KUKA KRL program: EPS_2_25748_MH04A_A_20260121065900.src

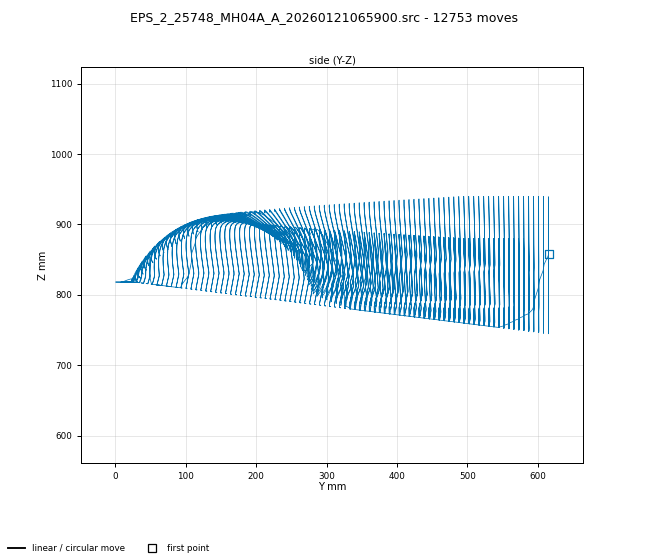
[picture p0: tool path of EPS_2_25748_MH04A_A_20260121065900.src, 12753 of 12755 moves have a stored position in this frame; points joined in program order, loops and branches not executed]
&ACCESS RVP
&REL 4
&COMMENT QRS 19112012
&PARAM EDITMASK = *
DEF PART()
EXT BAS (BAS_COMMAND :IN,REAL :IN )
INT I
BAS (#INITMOV,0 )

;KUKA QRS Post kuka4.cps  Date:22-06-2017 !

File_ID=3002

QRS_PRE_INIT()

;Init var - Until changes are made in qrs_pre_init
Outlet_Square_prg=0
Inlet_1_Square_prg=0
Inlet_2_Square_prg=0
Inlet_3_Square_prg=0
Inlet_4_Square_prg=0
Inlet_5_Square_prg=0

Outlet_1={X 0.000, Y 493.160, Z 839.500, B 0.000, E1 0.000 }
Inlet_1={X 0.000, Y 497.530, Z 779.500, B 0.000, E1 90.000 }
Inlet_2={X 0.000, Y 497.530, Z 779.500, B 0.000, E1 270.000 }
Outlet_1_type=201
Inlet_1_type=201
Inlet_2_type=201
;QRS#1=Sidecore dimensions
;QRS#2=200-8" PVC SDR 35
;QRS#3=200-8" PVC SDR 35
;QRS#4=200-8" PVC SDR 35
;QRS#5=
;QRS#6=
;QRS#7=
;QRS#8=
;QRS#9=12-08 PSX
;QRS#10=12-08 PSX
;QRS#11=12-08 PSX
;QRS#12=
;QRS#13=
;QRS#14=
;QRS#15=
;QRS#16=1220x127x1219 4'
;QRS#17=EPS Height
;QRS#18=940
;QRS#19=*
;QRS#20= UPDATED VERSION 22-06-2017
;QRS#21=*
Outlet_Square=0100
Inlet_1_Square=0100
Inlet_2_Square=0100
Inlet_3_Square=0
Inlet_4_Square=0
Inlet_5_Square=0
Mill_Square=1
Outlet_Square_Prg=204
Inlet_1_Square_prg=204
Inlet_2_Square_prg=204

QRS_INIT()

$ADVANCE=5

; T1
PTP {E1 173.418,E2 173.418}
PTP {X 0,Y 615.496,A -85,B 0,C 180,E1 173.418,E2 173.418,E3 0,E4 0,E5 0,E6 0}
QRS_SPEED_INIT()
LIN {X 0,Y 615.496,Z 858.208,A -85,B 0,C 180,E1 173.418,E2 173.418,E3 0,E4 0,E5 0,E6 0} C_VEL
LIN {X 0,Y 615.497,Z 850.543,A -85,B 0,C 180,E1 172.455,E2 172.455} C_VEL
LIN {X 0,Y 615.498,Z 840.767,A -85,B 0,C 180,E1 171.464,E2 171.464} C_VEL
LIN {X 0,Y 615.498,Z 830.503,A -85,B 0,C 180,E1 170.636,E2 170.636} C_VEL
LIN {X 0,Y 615.496,Z 818.942,A -85,B 0,C 180,E1 169.89,E2 169.89} C_VEL
LIN {X 0,Y 615.451,Z 807.364,A -85,B 0,C 180,E1 169.304,E2 169.304} C_VEL
LIN {X 0,Y 615.447,Z 795.462,A -85,B 0,C 180,E1 168.848,E2 168.848} C_VEL
LIN {X 0,Y 615.479,Z 783.419,A -85,B 0,C 180,E1 168.516,E2 168.516} C_VEL
LIN {X 0,Y 615.492,Z 776.192,A -85,B 0,C 180,E1 168.37,E2 168.37} C_VEL
LIN {X 0,Y 615.47,Z 772.045,A -85,B 0,C 180,E1 165.451,E2 165.451} C_VEL
LIN {X 0,Y 615.475,Z 768.231,A -85,B 0,C 180,E1 162.73,E2 162.73} C_VEL
LIN {X 0,Y 615.494,Z 764.414,A -85,B 0,C 180,E1 159.968,E2 159.968} C_VEL
LIN {X 0,Y 615.496,Z 761.258,A -85,B 0,C 180,E1 157.653,E2 157.653} C_VEL
LIN {X 0,Y 615.471,Z 757.73,A -85,B 0,C 180,E1 155.008,E2 155.008} C_VEL
LIN {X 0,Y 615.479,Z 754.866,A -85,B 0,C 180,E1 152.823,E2 152.823} C_VEL
LIN {X 0,Y 615.474,Z 751.515,A -85,B 0,C 180,E1 150.208,E2 150.208} C_VEL
LIN {X 0,Y 615.499,Z 748.171,A -85,B 0,C 180,E1 147.544,E2 147.544} C_VEL
LIN {X 0,Y 615.496,Z 745.306,A -85,B 0,C 180,E1 145.187,E2 145.187} C_VEL
LIN {X 0,Y 615.457,Z 744.691,A -85,B 0,C 180,E1 144.171,E2 144.171} C_VEL
LIN {X 0,Y 615.461,Z 744.688,A -85,B 0,C 180,E1 141.931,E2 141.931} C_VEL
LIN {X 0,Y 615.487,Z 744.683,A -85,B 0,C 180,E1 139.395,E2 139.395} C_VEL
LIN {X 0,Y 615.495,Z 744.698,A -85,B 0,C 180,E1 136.757,E2 136.757} C_VEL
LIN {X 0,Y 615.452,Z 744.692,A -85,B 0,C 180,E1 133.995,E2 133.995} C_VEL
LIN {X 0,Y 615.465,Z 744.686,A -85,B 0,C 180,E1 131.476,E2 131.476} C_VEL
LIN {X 0,Y 615.498,Z 744.688,A -85,B 0,C 180,E1 128.904,E2 128.904} C_VEL
LIN {X 0,Y 615.478,Z 744.701,A -85,B 0,C 180,E1 126.426,E2 126.426} C_VEL
LIN {X 0,Y 615.453,Z 744.696,A -85,B 0,C 180,E1 124.024,E2 124.024} C_VEL
LIN {X 0,Y 615.441,Z 744.693,A -85,B 0,C 180,E1 121.688,E2 121.688} C_VEL
LIN {X 0,Y 615.44,Z 744.692,A -85,B 0,C 180,E1 119.409,E2 119.409} C_VEL
LIN {X 0,Y 615.46,Z 744.69,A -85,B 0,C 180,E1 117.042,E2 117.042} C_VEL
LIN {X 0,Y 615.458,Z 744.698,A -85,B 0,C 180,E1 114.005,E2 114.005} C_VEL
LIN {X 0,Y 615.431,Z 744.694,A -85,B 0,C 180,E1 111.434,E2 111.434} C_VEL
LIN {X 0,Y 615.429,Z 744.695,A -85,B 0,C 180,E1 109.34,E2 109.34} C_VEL
LIN {X 0,Y 615.475,Z 744.692,A -85,B 0,C 180,E1 106.587,E2 106.587} C_VEL
LIN {X 0,Y 615.458,Z 744.699,A -85,B 0,C 180,E1 103.875,E2 103.875} C_VEL
LIN {X 0,Y 615.42,Z 744.697,A -85,B 0,C 180,E1 101.194,E2 101.194} C_VEL
LIN {X 0,Y 615.455,Z 744.695,A -85,B 0,C 180,E1 98.537,E2 98.537} C_VEL
LIN {X 0,Y 615.475,Z 744.7,A -85,B 0,C 180,E1 95.899,E2 95.899} C_VEL
LIN {X 0,Y 615.416,Z 744.699,A -85,B 0,C 180,E1 93.273,E2 93.273} C_VEL
LIN {X 0,Y 615.418,Z 744.699,A -85,B 0,C 180,E1 91.309,E2 91.309} C_VEL
LIN {X 0,Y 615.421,Z 744.7,A -85,B 0,C 180,E1 89.346,E2 89.346} C_VEL
LIN {X 0,Y 615.426,Z 744.7,A -85,B 0,C 180,E1 87.382,E2 87.382} C_VEL
LIN {X 0,Y 615.432,Z 744.7,A -85,B 0,C 180,E1 85.415,E2 85.415} C_VEL
LIN {X 0,Y 615.442,Z 744.699,A -85,B 0,C 180,E1 83.443,E2 83.443} C_VEL
LIN {X 0,Y 615.41,Z 744.699,A -85,B 0,C 180,E1 80.8,E2 80.8} C_VEL
LIN {X 0,Y 615.412,Z 744.698,A -85,B 0,C 180,E1 78.805,E2 78.805} C_VEL
LIN {X 0,Y 615.415,Z 744.698,A -85,B 0,C 180,E1 76.797,E2 76.797} C_VEL
LIN {X 0,Y 615.418,Z 744.697,A -85,B 0,C 180,E1 74.772,E2 74.772} C_VEL
LIN {X 0,Y 615.42,Z 744.696,A -85,B 0,C 180,E1 72.727,E2 72.727} C_VEL
LIN {X 0,Y 615.422,Z 744.696,A -85,B 0,C 180,E1 70.66,E2 70.66} C_VEL
LIN {X 0,Y 615.422,Z 744.696,A -85,B 0,C 180,E1 68.566,E2 68.566} C_VEL
LIN {X 0,Y 615.446,Z 744.698,A -85,B 0,C 180,E1 65.998,E2 65.998} C_VEL
LIN {X 0,Y 615.458,Z 744.692,A -85,B 0,C 180,E1 62.958,E2 62.958} C_VEL
LIN {X 0,Y 615.438,Z 744.693,A -85,B 0,C 180,E1 60.591,E2 60.591} C_VEL
LIN {X 0,Y 615.434,Z 744.694,A -85,B 0,C 180,E1 58.311,E2 58.311} C_VEL
LIN {X 0,Y 615.441,Z 744.696,A -85,B 0,C 180,E1 55.975,E2 55.975} C_VEL
LIN {X 0,Y 615.497,Z 744.689,A -85,B 0,C 180,E1 53.061,E2 53.061} C_VEL
LIN {X 0,Y 615.443,Z 744.691,A -85,B 0,C 180,E1 50.246,E2 50.246} C_VEL
LIN {X 0,Y 615.461,Z 744.697,A -85,B 0,C 180,E1 47.645,E2 47.645} C_VEL
LIN {X 0,Y 615.497,Z 744.689,A -85,B 0,C 180,E1 44.932,E2 44.932} C_VEL
LIN {X 0,Y 615.465,Z 744.687,A -85,B 0,C 180,E1 42.354,E2 42.354} C_VEL
LIN {X 0,Y 615.453,Z 744.693,A -85,B 0,C 180,E1 39.752,E2 39.752} C_VEL
LIN {X 0,Y 615.492,Z 744.694,A -85,B 0,C 180,E1 36.937,E2 36.937} C_VEL
LIN {X 0,Y 615.458,Z 744.693,A -85,B 0,C 180,E1 35.617,E2 35.617} C_VEL
LIN {X 0,Y 615.494,Z 745.333,A -85,B 0,C 180,E1 34.701,E2 34.701} C_VEL
LIN {X 0,Y 615.492,Z 748.215,A -85,B 0,C 180,E1 32.331,E2 32.331} C_VEL
LIN {X 0,Y 615.47,Z 751.401,A -85,B 0,C 180,E1 29.791,E2 29.791} C_VEL
LIN {X 0,Y 615.486,Z 754.919,A -85,B 0,C 180,E1 27.044,E2 27.044} C_VEL
LIN {X 0,Y 615.495,Z 758.56,A -85,B 0,C 180,E1 24.271,E2 24.271} C_VEL
LIN {X 0,Y 615.492,Z 762.386,A -85,B 0,C 180,E1 21.431,E2 21.431} C_VEL
LIN {X 0,Y 615.476,Z 766.256,A -85,B 0,C 180,E1 18.601,E2 18.601} C_VEL
LIN {X 0,Y 615.492,Z 770.016,A -85,B 0,C 180,E1 15.904,E2 15.904} C_VEL
LIN {X 0,Y 615.469,Z 773.827,A -85,B 0,C 180,E1 13.201,E2 13.201} C_VEL
LIN {X 0,Y 615.49,Z 776.183,A -85,B 0,C 180,E1 11.547,E2 11.547} C_VEL
LIN {X 0,Y 615.462,Z 791.288,A -85,B 0,C 180,E1 11.193,E2 11.193} C_VEL
LIN {X 0,Y 615.447,Z 803.206,A -85,B 0,C 180,E1 10.782,E2 10.782} C_VEL
LIN {X 0,Y 615.492,Z 815.77,A -85,B 0,C 180,E1 10.194,E2 10.194} C_VEL
LIN {X 0,Y 615.499,Z 826.859,A -85,B 0,C 180,E1 9.529,E2 9.529} C_VEL
LIN {X 0,Y 615.498,Z 835.832,A -85,B 0,C 180,E1 8.867,E2 8.867} C_VEL
LIN {X 0,Y 615.498,Z 845.041,A -85,B 0,C 180,E1 8.04,E2 8.04} C_VEL
LIN {X 0,Y 615.499,Z 853.896,A -85,B 0,C 180,E1 7.057,E2 7.057} C_VEL
LIN {X 0,Y 615.497,Z 861.128,A -85,B 0,C 180,E1 6.062,E2 6.062} C_VEL
LIN {X 0,Y 615.497,Z 865.962,A -85,B 0,C 180,E1 5.24,E2 5.24} C_VEL
LIN {X 0,Y 615.493,Z 870.661,A -85,B 0,C 180,E1 4.256,E2 4.256} C_VEL
LIN {X 0,Y 615.495,Z 874.257,A -85,B 0,C 180,E1 3.272,E2 3.272} C_VEL
LIN {X 0,Y 615.496,Z 876.117,A -85,B 0,C 180,E1 2.617,E2 2.617} C_VEL
LIN {X 0,Y 615.497,Z 877.535,A -85,B 0,C 180,E1 1.962,E2 1.962} C_VEL
LIN {X 0,Y 615.496,Z 879.142,A -85,B 0,C 180,E1 0.654,E2 0.654} C_VEL
LIN {X 0,Y 615.494,Z 879.384,A -85,B 0,C 180,E1 -0.001,E2 -0.001} C_VEL
LIN {X 0,Y 615.496,Z 879.205,A -85,B 0,C 180,E1 -0.655,E2 -0.655} C_VEL
LIN {X 0,Y 615.496,Z 877.682,A -85,B 0,C 180,E1 -1.964,E2 -1.964} C_VEL
LIN {X 0,Y 615.498,Z 876.34,A -85,B 0,C 180,E1 -2.618,E2 -2.618} C_VEL
LIN {X 0,Y 615.496,Z 873.492,A -85,B 0,C 180,E1 -3.601,E2 -3.601} C_VEL
LIN {X 0,Y 615.498,Z 869.631,A -85,B 0,C 180,E1 -4.585,E2 -4.585} C_VEL
LIN {X 0,Y 615.498,Z 864.648,A -85,B 0,C 180,E1 -5.57,E2 -5.57} C_VEL
LIN {X 0,Y 615.496,Z 858.207,A -85,B 0,C 180,E1 -6.583,E2 -6.583} C_VEL
LIN {X 0,Y 615.497,Z 850.531,A -85,B 0,C 180,E1 -7.546,E2 -7.546} C_VEL
LIN {X 0,Y 615.498,Z 840.752,A -85,B 0,C 180,E1 -8.537,E2 -8.537} C_VEL
LIN {X 0,Y 615.498,Z 830.484,A -85,B 0,C 180,E1 -9.365,E2 -9.365} C_VEL
LIN {X 0,Y 615.488,Z 818.92,A -85,B 0,C 180,E1 -10.112,E2 -10.112} C_VEL
LIN {X 0,Y 615.496,Z 807.057,A -85,B 0,C 180,E1 -10.708,E2 -10.708} C_VEL
LIN {X 0,Y 615.485,Z 794.142,A -85,B 0,C 180,E1 -11.194,E2 -11.194} C_VEL
LIN {X 0,Y 615.486,Z 781.533,A -85,B 0,C 180,E1 -11.527,E2 -11.527} C_VEL
LIN {X 0,Y 615.487,Z 776.191,A -85,B 0,C 180,E1 -11.632,E2 -11.632} C_VEL
LIN {X 0,Y 615.492,Z 772.038,A -85,B 0,C 180,E1 -14.55,E2 -14.55} C_VEL
LIN {X 0,Y 615.494,Z 768.225,A -85,B 0,C 180,E1 -17.271,E2 -17.271} C_VEL
LIN {X 0,Y 615.46,Z 764.418,A -85,B 0,C 180,E1 -20.034,E2 -20.034} C_VEL
LIN {X 0,Y 615.482,Z 761.265,A -85,B 0,C 180,E1 -22.344,E2 -22.344} C_VEL
LIN {X 0,Y 615.491,Z 757.724,A -85,B 0,C 180,E1 -24.992,E2 -24.992} C_VEL
LIN {X 0,Y 615.488,Z 754.863,A -85,B 0,C 180,E1 -27.178,E2 -27.178} C_VEL
LIN {X 0,Y 615.46,Z 751.521,A -85,B 0,C 180,E1 -29.79,E2 -29.79} C_VEL
LIN {X 0,Y 615.473,Z 748.173,A -85,B 0,C 180,E1 -32.459,E2 -32.459} C_VEL
LIN {X 0,Y 615.497,Z 745.304,A -85,B 0,C 180,E1 -34.815,E2 -34.815} C_VEL
LIN {X 0,Y 615.468,Z 744.69,A -85,B 0,C 180,E1 -35.831,E2 -35.831} C_VEL
LIN {X 0,Y 615.461,Z 744.689,A -85,B 0,C 180,E1 -38.071,E2 -38.071} C_VEL
LIN {X 0,Y 615.471,Z 744.692,A -85,B 0,C 180,E1 -40.608,E2 -40.608} C_VEL
LIN {X 0,Y 615.492,Z 744.695,A -85,B 0,C 180,E1 -43.245,E2 -43.245} C_VEL
LIN {X 0,Y 615.479,Z 744.684,A -85,B 0,C 180,E1 -46.004,E2 -46.004} C_VEL
LIN {X 0,Y 615.485,Z 744.702,A -85,B 0,C 180,E1 -48.906,E2 -48.906} C_VEL
LIN {X 0,Y 615.488,Z 744.696,A -85,B 0,C 180,E1 -51.095,E2 -51.095} C_VEL
LIN {X 0,Y 615.484,Z 744.685,A -85,B 0,C 180,E1 -53.575,E2 -53.575} C_VEL
LIN {X 0,Y 615.485,Z 744.816,A -85,B 0,C 180,E1 -54.535,E2 -54.535} C_VEL
LIN {X 0,Y 615.482,Z 753.576,A -85,B 0,C 180,E1 -57.154,E2 -57.154} C_VEL
LIN {X 0,Y 615.482,Z 762.831,A -85,B 0,C 180,E1 -59.839,E2 -59.839} C_VEL
LIN {X 0,Y 615.494,Z 772.075,A -85,B 0,C 180,E1 -62.455,E2 -62.455} C_VEL
LIN {X 0,Y 615.47,Z 781.315,A -85,B 0,C 180,E1 -65.007,E2 -65.007} C_VEL
LIN {X 0,Y 615.489,Z 791.092,A -85,B 0,C 180,E1 -67.654,E2 -67.654} C_VEL
LIN {X 0,Y 615.487,Z 801.099,A -85,B 0,C 180,E1 -70.315,E2 -70.315} C_VEL
LIN {X 0,Y 615.469,Z 811.641,A -85,B 0,C 180,E1 -73.071,E2 -73.071} C_VEL
LIN {X 0,Y 615.486,Z 822.077,A -85,B 0,C 180,E1 -75.761,E2 -75.761} C_VEL
LIN {X 0,Y 615.482,Z 832.208,A -85,B 0,C 180,E1 -78.348,E2 -78.348} C_VEL
LIN {X 0,Y 615.498,Z 846.819,A -85,B 0,C 180,E1 -78.64,E2 -78.64} C_VEL
LIN {X 0,Y 615.476,Z 859.709,A -85,B 0,C 180,E1 -79.042,E2 -79.042} C_VEL
LIN {X 0,Y 615.482,Z 871.766,A -85,B 0,C 180,E1 -79.556,E2 -79.556} C_VEL
LIN {X 0,Y 615.48,Z 882.389,A -85,B 0,C 180,E1 -80.138,E2 -80.138} C_VEL
LIN {X 0,Y 615.498,Z 893.231,A -85,B 0,C 180,E1 -80.884,E2 -80.884} C_VEL
LIN {X 0,Y 615.497,Z 903.811,A -85,B 0,C 180,E1 -81.794,E2 -81.794} C_VEL
LIN {X 0,Y 615.498,Z 911.606,A -85,B 0,C 180,E1 -82.62,E2 -82.62} C_VEL
LIN {X 0,Y 615.496,Z 919.203,A -85,B 0,C 180,E1 -83.608,E2 -83.608} C_VEL
LIN {X 0,Y 615.498,Z 926.204,A -85,B 0,C 180,E1 -84.759,E2 -84.759} C_VEL
LIN {X 0,Y 615.493,Z 930.851,A -85,B 0,C 180,E1 -85.744,E2 -85.744} C_VEL
LIN {X 0,Y 615.496,Z 934.398,A -85,B 0,C 180,E1 -86.727,E2 -86.727} C_VEL
LIN {X 0,Y 615.497,Z 936.233,A -85,B 0,C 180,E1 -87.382,E2 -87.382} C_VEL
LIN {X 0,Y 615.496,Z 937.608,A -85,B 0,C 180,E1 -88.037,E2 -88.037} C_VEL
LIN {X 0,Y 615.496,Z 939.174,A -85,B 0,C 180,E1 -89.346,E2 -89.346} C_VEL
LIN {X 0,Y 615.494,Z 939.389,A -85,B 0,C 180,E1 -90,E2 -90} C_VEL
LIN {X 0,Y 615.496,Z 938.58,A -85,B 0,C 180,E1 -91.309,E2 -91.309} C_VEL
LIN {X 0,Y 615.496,Z 937.608,A -85,B 0,C 180,E1 -91.963,E2 -91.963} C_VEL
LIN {X 0,Y 615.497,Z 936.233,A -85,B 0,C 180,E1 -92.618,E2 -92.618} C_VEL
LIN {X 0,Y 615.496,Z 933.349,A -85,B 0,C 180,E1 -93.601,E2 -93.601} C_VEL
LIN {X 0,Y 615.498,Z 929.441,A -85,B 0,C 180,E1 -94.584,E2 -94.584} C_VEL
LIN {X 0,Y 615.499,Z 924.405,A -85,B 0,C 180,E1 -95.57,E2 -95.57} C_VEL
LIN {X 0,Y 615.497,Z 917.87,A -85,B 0,C 180,E1 -96.583,E2 -96.583} C_VEL
LIN {X 0,Y 615.497,Z 910.133,A -85,B 0,C 180,E1 -97.545,E2 -97.545} C_VEL
LIN {X 0,Y 615.498,Z 902.044,A -85,B 0,C 180,E1 -98.371,E2 -98.371} C_VEL
LIN {X 0,Y 615.499,Z 892.167,A -85,B 0,C 180,E1 -99.199,E2 -99.199} C_VEL
LIN {X 0,Y 615.482,Z 880.981,A -85,B 0,C 180,E1 -99.945,E2 -99.945} C_VEL
LIN {X 0,Y 615.478,Z 870.023,A -85,B 0,C 180,E1 -100.527,E2 -100.527} C_VEL
LIN {X 0,Y 615.479,Z 857.592,A -85,B 0,C 180,E1 -101.037,E2 -101.037} C_VEL
LIN {X 0,Y 615.497,Z 845.06,A -85,B 0,C 180,E1 -101.401,E2 -101.401} C_VEL
LIN {X 0,Y 615.482,Z 832.208,A -85,B 0,C 180,E1 -101.652,E2 -101.652} C_VEL
LIN {X 0,Y 615.486,Z 822.077,A -85,B 0,C 180,E1 -104.239,E2 -104.239} C_VEL
LIN {X 0,Y 615.469,Z 811.641,A -85,B 0,C 180,E1 -106.929,E2 -106.929} C_VEL
LIN {X 0,Y 615.487,Z 801.099,A -85,B 0,C 180,E1 -109.685,E2 -109.685} C_VEL
LIN {X 0,Y 615.489,Z 791.092,A -85,B 0,C 180,E1 -112.346,E2 -112.346} C_VEL
LIN {X 0,Y 615.47,Z 781.315,A -85,B 0,C 180,E1 -114.993,E2 -114.993} C_VEL
LIN {X 0,Y 615.494,Z 772.075,A -85,B 0,C 180,E1 -117.545,E2 -117.545} C_VEL
LIN {X 0,Y 615.482,Z 762.831,A -85,B 0,C 180,E1 -120.161,E2 -120.161} C_VEL
LIN {X 0,Y 615.482,Z 753.576,A -85,B 0,C 180,E1 -122.846,E2 -122.846} C_VEL
LIN {X 0,Y 615.484,Z 744.692,A -85,B 0,C 180,E1 -125.516,E2 -125.516} C_VEL
LIN {X 0,Y 615.489,Z 744.682,A -85,B 0,C 180,E1 -128.069,E2 -128.069} C_VEL
LIN {X 0,Y 615.486,Z 744.688,A -85,B 0,C 180,E1 -130.607,E2 -130.607} C_VEL
LIN {X 0,Y 615.482,Z 744.697,A -85,B 0,C 180,E1 -133.245,E2 -133.245} C_VEL
LIN {X 0,Y 615.474,Z 744.685,A -85,B 0,C 180,E1 -136.004,E2 -136.004} C_VEL
LIN {X 0,Y 615.491,Z 744.7,A -85,B 0,C 180,E1 -138.905,E2 -138.905} C_VEL
LIN {X 0,Y 615.491,Z 744.696,A -85,B 0,C 180,E1 -141.095,E2 -141.095} C_VEL
LIN {X 0,Y 615.466,Z 744.69,A -85,B 0,C 180,E1 -143.573,E2 -143.573} C_VEL
LIN {X 0,Y 615.486,Z 744.688,A -85,B 0,C 180,E1 -144.384,E2 -144.384} C_VEL
LIN {X 0,Y 615.486,Z 745.336,A -85,B 0,C 180,E1 -145.3,E2 -145.3} C_VEL
LIN {X 0,Y 615.465,Z 748.227,A -85,B 0,C 180,E1 -147.673,E2 -147.673} C_VEL
LIN {X 0,Y 615.461,Z 751.405,A -85,B 0,C 180,E1 -150.21,E2 -150.21} C_VEL
LIN {X 0,Y 615.491,Z 754.917,A -85,B 0,C 180,E1 -152.955,E2 -152.955} C_VEL
LIN {X 0,Y 615.472,Z 758.562,A -85,B 0,C 180,E1 -155.727,E2 -155.727} C_VEL
LIN {X 0,Y 615.465,Z 761.428,A -85,B 0,C 180,E1 -157.862,E2 -157.862} C_VEL
LIN {X 0,Y 615.488,Z 765.243,A -85,B 0,C 180,E1 -160.662,E2 -160.662} C_VEL
LIN {X 0,Y 615.494,Z 769.267,A -85,B 0,C 180,E1 -163.568,E2 -163.568} C_VEL
LIN {X 0,Y 615.463,Z 772.883,A -85,B 0,C 180,E1 -166.125,E2 -166.125} C_VEL
LIN {X 0,Y 615.48,Z 776.183,A -85,B 0,C 180,E1 -168.452,E2 -168.452} C_VEL
LIN {X 0,Y 615.488,Z 791.234,A -85,B 0,C 180,E1 -168.806,E2 -168.806} C_VEL
LIN {X 0,Y 615.498,Z 803.861,A -85,B 0,C 180,E1 -169.247,E2 -169.247} C_VEL
LIN {X 0,Y 615.49,Z 815.745,A -85,B 0,C 180,E1 -169.805,E2 -169.805} C_VEL
LIN {X 0,Y 615.497,Z 826.838,A -85,B 0,C 180,E1 -170.469,E2 -170.469} C_VEL
LIN {X 0,Y 615.498,Z 835.815,A -85,B 0,C 180,E1 -171.132,E2 -171.132} C_VEL
LIN {X 0,Y 615.498,Z 845.028,A -85,B 0,C 180,E1 -171.959,E2 -171.959} C_VEL
LIN {X 0,Y 615.499,Z 853.888,A -85,B 0,C 180,E1 -172.942,E2 -172.942} C_VEL
LIN {X 0,Y 615.497,Z 861.119,A -85,B 0,C 180,E1 -173.936,E2 -173.936} C_VEL
LIN {X 0,Y 615.497,Z 865.955,A -85,B 0,C 180,E1 -174.758,E2 -174.758} C_VEL
LIN {X 0,Y 615.494,Z 870.655,A -85,B 0,C 180,E1 -175.743,E2 -175.743} C_VEL
LIN {X 0,Y 615.494,Z 874.252,A -85,B 0,C 180,E1 -176.726,E2 -176.726} C_VEL
LIN {X 0,Y 615.498,Z 876.112,A -85,B 0,C 180,E1 -177.382,E2 -177.382} C_VEL
LIN {X 0,Y 615.497,Z 877.532,A -85,B 0,C 180,E1 -178.036,E2 -178.036} C_VEL
LIN {X 0,Y 615.497,Z 879.141,A -85,B 0,C 180,E1 -179.345,E2 -179.345} C_VEL
LIN {X 0,Y 615.494,Z 879.384,A -85,B 0,C 180,E1 -179.999,E2 -179.999} C_VEL
LIN {X 0,Y 615.495,Z 879.206,A -85,B 0,C 180,E1 -180.654,E2 -180.654} C_VEL
LIN {X 0,Y 615.497,Z 877.684,A -85,B 0,C 180,E1 -181.962,E2 -181.962} C_VEL
LIN {X 0,Y 615.498,Z 876.343,A -85,B 0,C 180,E1 -182.617,E2 -182.617} C_VEL
LIN {X 0,Y 615.497,Z 873.496,A -85,B 0,C 180,E1 -183.6,E2 -183.6} C_VEL
LIN {X 0,Y 615.498,Z 869.637,A -85,B 0,C 180,E1 -184.584,E2 -184.584} C_VEL
LIN {X 0,Y 615.498,Z 864.655,A -85,B 0,C 180,E1 -185.569,E2 -185.569} C_VEL
LIN {X 0,Y 615.496,Z 858.208,A -85,B 0,C 180,E1 -186.582,E2 -186.582} C_VEL
LIN {X 0,Y 614.829,Z 855.026,A -85,B 0,C 180,E1 -187.031,E2 -187.031} C_VEL
LIN {X 0,Y 611.989,Z 849.453,A -85,B 0,C 180,E1 -187.748,E2 -187.748} C_VEL
LIN {X 0,Y 609.138,Z 843.177,A -85,B 0,C 180,E1 -188.429,E2 -188.429} C_VEL
LIN {X 0,Y 608.477,Z 838.936,A -85,B 0,C 180,E1 -188.819,E2 -188.819} C_VEL
LIN {X 0,Y 608.498,Z 828.401,A -85,B 0,C 180,E1 -189.64,E2 -189.64} C_VEL
LIN {X 0,Y 608.49,Z 817.625,A -85,B 0,C 180,E1 -190.312,E2 -190.312} C_VEL
LIN {X 0,Y 608.48,Z 805.618,A -85,B 0,C 180,E1 -190.9,E2 -190.9} C_VEL
LIN {X 0,Y 608.505,Z 792.99,A -85,B 0,C 180,E1 -191.365,E2 -191.365} C_VEL
LIN {X 0,Y 608.556,Z 780.698,A -85,B 0,C 180,E1 -191.68,E2 -191.68} C_VEL
LIN {X 0,Y 608.443,Z 776.675,A -85,B 0,C 180,E1 -191.767,E2 -191.767} C_VEL
LIN {X 0,Y 608.401,Z 772.5,A -85,B 0,C 180,E1 -194.722,E2 -194.722} C_VEL
LIN {X 0,Y 608.406,Z 769.616,A -85,B 0,C 180,E1 -196.785,E2 -196.785} C_VEL
LIN {X 0,Y 608.412,Z 765.771,A -85,B 0,C 180,E1 -199.571,E2 -199.571} C_VEL
LIN {X 0,Y 608.428,Z 761.842,A -85,B 0,C 180,E1 -202.468,E2 -202.468} C_VEL
LIN {X 0,Y 608.424,Z 758.08,A -85,B 0,C 180,E1 -205.301,E2 -205.301} C_VEL
LIN {X 0,Y 608.435,Z 754.234,A -85,B 0,C 180,E1 -208.266,E2 -208.266} C_VEL
LIN {X 0,Y 608.429,Z 751.349,A -85,B 0,C 180,E1 -210.546,E2 -210.546} C_VEL
LIN {X 0,Y 608.43,Z 748.465,A -85,B 0,C 180,E1 -212.88,E2 -212.88} C_VEL
LIN {X 0,Y 608.405,Z 745.703,A -85,B 0,C 180,E1 -215.279,E2 -215.279} C_VEL
LIN {X 0,Y 608.454,Z 745.689,A -85,B 0,C 180,E1 -217.746,E2 -217.746} C_VEL
LIN {X 0,Y 608.438,Z 745.689,A -85,B 0,C 180,E1 -220.327,E2 -220.327} C_VEL
LIN {X 0,Y 608.479,Z 745.695,A -85,B 0,C 180,E1 -223.309,E2 -223.309} C_VEL
LIN {X 0,Y 608.445,Z 745.688,A -85,B 0,C 180,E1 -226.128,E2 -226.128} C_VEL
LIN {X 0,Y 608.454,Z 745.688,A -85,B 0,C 180,E1 -228.823,E2 -228.823} C_VEL
LIN {X 0,Y 608.444,Z 745.694,A -85,B 0,C 180,E1 -231.761,E2 -231.761} C_VEL
LIN {X 0,Y 608.43,Z 745.693,A -85,B 0,C 180,E1 -233.955,E2 -233.955} C_VEL
LIN {X 0,Y 608.434,Z 745.689,A -85,B 0,C 180,E1 -236.327,E2 -236.327} C_VEL
LIN {X 0,Y 608.434,Z 745.689,A -85,B 0,C 180,E1 -238.732,E2 -238.732} C_VEL
LIN {X 0,Y 608.446,Z 745.697,A -85,B 0,C 180,E1 -241.733,E2 -241.733} C_VEL
LIN {X 0,Y 608.43,Z 745.691,A -85,B 0,C 180,E1 -244.285,E2 -244.285} C_VEL
LIN {X 0,Y 608.419,Z 745.691,A -85,B 0,C 180,E1 -246.875,E2 -246.875} C_VEL
LIN {X 0,Y 608.454,Z 745.698,A -85,B 0,C 180,E1 -249.725,E2 -249.725} C_VEL
LIN {X 0,Y 608.432,Z 745.7,A -85,B 0,C 180,E1 -251.828,E2 -251.828} C_VEL
LIN {X 0,Y 608.445,Z 745.697,A -85,B 0,C 180,E1 -253.906,E2 -253.906} C_VEL
LIN {X 0,Y 608.411,Z 745.692,A -85,B 0,C 180,E1 -256.642,E2 -256.642} C_VEL
LIN {X 0,Y 608.431,Z 745.692,A -85,B 0,C 180,E1 -259.35,E2 -259.35} C_VEL
LIN {X 0,Y 608.459,Z 745.695,A -85,B 0,C 180,E1 -262.033,E2 -262.033} C_VEL
LIN {X 0,Y 608.404,Z 745.694,A -85,B 0,C 180,E1 -264.698,E2 -264.698} C_VEL
LIN {X 0,Y 608.421,Z 745.692,A -85,B 0,C 180,E1 -267.352,E2 -267.352} C_VEL
LIN {X 0,Y 608.467,Z 745.696,A -85,B 0,C 180,E1 -270,E2 -270} C_VEL
LIN {X 0,Y 608.42,Z 745.693,A -85,B 0,C 180,E1 -272.648,E2 -272.648} C_VEL
LIN {X 0,Y 608.394,Z 745.694,A -85,B 0,C 180,E1 -275.303,E2 -275.303} C_VEL
LIN {X 0,Y 608.42,Z 745.698,A -85,B 0,C 180,E1 -277.968,E2 -277.968} C_VEL
LIN {X 0,Y 608.394,Z 745.695,A -85,B 0,C 180,E1 -280.925,E2 -280.925} C_VEL
LIN {X 0,Y 608.403,Z 745.693,A -85,B 0,C 180,E1 -283.358,E2 -283.358} C_VEL
LIN {X 0,Y 608.415,Z 745.692,A -85,B 0,C 180,E1 -285.407,E2 -285.407} C_VEL
LIN {X 0,Y 608.401,Z 745.693,A -85,B 0,C 180,E1 -287.478,E2 -287.478} C_VEL
LIN {X 0,Y 608.404,Z 745.693,A -85,B 0,C 180,E1 -289.572,E2 -289.572} C_VEL
LIN {X 0,Y 608.422,Z 745.692,A -85,B 0,C 180,E1 -291.693,E2 -291.693} C_VEL
LIN {X 0,Y 608.438,Z 745.697,A -85,B 0,C 180,E1 -294.572,E2 -294.572} C_VEL
LIN {X 0,Y 608.412,Z 745.692,A -85,B 0,C 180,E1 -297.52,E2 -297.52} C_VEL
LIN {X 0,Y 608.426,Z 745.693,A -85,B 0,C 180,E1 -299.967,E2 -299.967} C_VEL
LIN {X 0,Y 608.443,Z 745.693,A -85,B 0,C 180,E1 -302.881,E2 -302.881} C_VEL
LIN {X 0,Y 608.422,Z 745.692,A -85,B 0,C 180,E1 -305.279,E2 -305.279} C_VEL
LIN {X 0,Y 608.438,Z 745.689,A -85,B 0,C 180,E1 -307.749,E2 -307.749} C_VEL
LIN {X 0,Y 608.427,Z 745.695,A -85,B 0,C 180,E1 -310.328,E2 -310.328} C_VEL
LIN {X 0,Y 608.478,Z 745.685,A -85,B 0,C 180,E1 -313.311,E2 -313.311} C_VEL
LIN {X 0,Y 608.441,Z 745.69,A -85,B 0,C 180,E1 -316.129,E2 -316.129} C_VEL
LIN {X 0,Y 608.455,Z 745.698,A -85,B 0,C 180,E1 -318.825,E2 -318.825} C_VEL
LIN {X 0,Y 608.447,Z 745.687,A -85,B 0,C 180,E1 -321.763,E2 -321.763} C_VEL
LIN {X 0,Y 608.436,Z 745.689,A -85,B 0,C 180,E1 -323.956,E2 -323.956} C_VEL
LIN {X 0,Y 608.429,Z 745.919,A -85,B 0,C 180,E1 -325.098,E2 -325.098} C_VEL
LIN {X 0,Y 608.419,Z 749.316,A -85,B 0,C 180,E1 -327.904,E2 -327.904} C_VEL
LIN {X 0,Y 608.42,Z 752.198,A -85,B 0,C 180,E1 -330.219,E2 -330.219} C_VEL
LIN {X 0,Y 608.427,Z 755.493,A -85,B 0,C 180,E1 -332.803,E2 -332.803} C_VEL
LIN {X 0,Y 608.425,Z 758.922,A -85,B 0,C 180,E1 -335.429,E2 -335.429} C_VEL
LIN {X 0,Y 608.422,Z 762.765,A -85,B 0,C 180,E1 -338.308,E2 -338.308} C_VEL
LIN {X 0,Y 608.415,Z 766.608,A -85,B 0,C 180,E1 -341.13,E2 -341.13} C_VEL
LIN {X 0,Y 608.428,Z 770.452,A -85,B 0,C 180,E1 -343.906,E2 -343.906} C_VEL
LIN {X 0,Y 608.419,Z 774.295,A -85,B 0,C 180,E1 -346.643,E2 -346.643} C_VEL
LIN {X 0,Y 608.444,Z 776.667,A -85,B 0,C 180,E1 -348.318,E2 -348.318} C_VEL
LIN {X 0,Y 608.52,Z 791.426,A -85,B 0,C 180,E1 -348.678,E2 -348.678} C_VEL
LIN {X 0,Y 608.481,Z 803.498,A -85,B 0,C 180,E1 -349.1,E2 -349.1} C_VEL
LIN {X 0,Y 608.491,Z 815.947,A -85,B 0,C 180,E1 -349.688,E2 -349.688} C_VEL
LIN {X 0,Y 608.499,Z 827.078,A -85,B 0,C 180,E1 -350.36,E2 -350.36} C_VEL
LIN {X 0,Y 608.474,Z 836.093,A -85,B 0,C 180,E1 -351.03,E2 -351.03} C_VEL
LIN {X 0,Y 608.464,Z 845.356,A -85,B 0,C 180,E1 -351.867,E2 -351.867} C_VEL
LIN {X 0,Y 608.466,Z 854.328,A -85,B 0,C 180,E1 -352.868,E2 -352.868} C_VEL
LIN {X 0,Y 608.444,Z 861.558,A -85,B 0,C 180,E1 -353.867,E2 -353.867} C_VEL
LIN {X 0,Y 608.462,Z 866.437,A -85,B 0,C 180,E1 -354.699,E2 -354.699} C_VEL
LIN {X 0,Y 608.439,Z 871.18,A -85,B 0,C 180,E1 -355.695,E2 -355.695} C_VEL
LIN {X 0,Y 608.425,Z 874.814,A -85,B 0,C 180,E1 -356.69,E2 -356.69} C_VEL
LIN {X 0,Y 608.425,Z 876.693,A -85,B 0,C 180,E1 -357.352,E2 -357.352} C_VEL
LIN {X 0,Y 608.442,Z 878.128,A -85,B 0,C 180,E1 -358.015,E2 -358.015} C_VEL
LIN {X 0,Y 608.439,Z 879.752,A -85,B 0,C 180,E1 -359.339,E2 -359.339} C_VEL
LIN {X 0,Y 608.434,Z 879.996,A -85,B 0,C 180,E1 -360.001,E2 -360.001} C_VEL
LIN {X 0,Y 608.439,Z 879.815,A -85,B 0,C 180,E1 -360.663,E2 -360.663} C_VEL
LIN {X 0,Y 608.441,Z 878.275,A -85,B 0,C 180,E1 -361.986,E2 -361.986} C_VEL
LIN {X 0,Y 608.427,Z 876.916,A -85,B 0,C 180,E1 -362.649,E2 -362.649} C_VEL
LIN {X 0,Y 608.449,Z 874.039,A -85,B 0,C 180,E1 -363.643,E2 -363.643} C_VEL
LIN {X 0,Y 608.433,Z 870.139,A -85,B 0,C 180,E1 -364.638,E2 -364.638} C_VEL
LIN {X 0,Y 608.449,Z 865.107,A -85,B 0,C 180,E1 -365.635,E2 -365.635} C_VEL
LIN {X 0,Y 608.441,Z 858.79,A -85,B 0,C 180,E1 -366.634,E2 -366.634} C_VEL
LIN {X 0,Y 608.476,Z 850.873,A -85,B 0,C 180,E1 -367.634,E2 -367.634} C_VEL
LIN {X 0,Y 608.472,Z 841.027,A -85,B 0,C 180,E1 -368.636,E2 -368.636} C_VEL
LIN {X 0,Y 608.48,Z 830.705,A -85,B 0,C 180,E1 -369.474,E2 -369.474} C_VEL
LIN {X 0,Y 608.485,Z 819.09,A -85,B 0,C 180,E1 -370.23,E2 -370.23} C_VEL
LIN {X 0,Y 608.517,Z 806.894,A -85,B 0,C 180,E1 -370.844,E2 -370.844} C_VEL
LIN {X 0,Y 608.527,Z 794.232,A -85,B 0,C 180,E1 -371.323,E2 -371.323} C_VEL
LIN {X 0,Y 608.539,Z 781.61,A -85,B 0,C 180,E1 -371.661,E2 -371.661} C_VEL
LIN {X 0,Y 608.43,Z 776.673,A -85,B 0,C 180,E1 -371.769,E2 -371.769} C_VEL
LIN {X 0,Y 608.419,Z 773.459,A -85,B 0,C 180,E1 -374.039,E2 -374.039} C_VEL
LIN {X 0,Y 608.421,Z 769.614,A -85,B 0,C 180,E1 -376.786,E2 -376.786} C_VEL
LIN {X 0,Y 608.408,Z 765.769,A -85,B 0,C 180,E1 -379.573,E2 -379.573} C_VEL
LIN {X 0,Y 608.438,Z 761.923,A -85,B 0,C 180,E1 -382.407,E2 -382.407} C_VEL
LIN {X 0,Y 608.423,Z 758.078,A -85,B 0,C 180,E1 -385.303,E2 -385.303} C_VEL
LIN {X 0,Y 608.414,Z 755.193,A -85,B 0,C 180,E1 -387.52,E2 -387.52} C_VEL
LIN {X 0,Y 608.427,Z 752.08,A -85,B 0,C 180,E1 -389.964,E2 -389.964} C_VEL
LIN {X 0,Y 608.417,Z 748.912,A -85,B 0,C 180,E1 -392.515,E2 -392.515} C_VEL
LIN {X 0,Y 608.435,Z 746.025,A -85,B 0,C 180,E1 -394.903,E2 -394.903} C_VEL
LIN {X 0,Y 608.419,Z 745.701,A -85,B 0,C 180,E1 -395.28,E2 -395.28} C_VEL
LIN {X 0,Y 608.459,Z 745.688,A -85,B 0,C 180,E1 -397.747,E2 -397.747} C_VEL
LIN {X 0,Y 608.437,Z 745.69,A -85,B 0,C 180,E1 -400.327,E2 -400.327} C_VEL
LIN {X 0,Y 608.456,Z 745.696,A -85,B 0,C 180,E1 -402.96,E2 -402.96} C_VEL
LIN {X 0,Y 608.462,Z 745.687,A -85,B 0,C 180,E1 -405.736,E2 -405.736} C_VEL
LIN {X 0,Y 608.455,Z 745.693,A -85,B 0,C 180,E1 -408.659,E2 -408.659} C_VEL
LIN {X 0,Y 608.469,Z 745.686,A -85,B 0,C 180,E1 -411.76,E2 -411.76} C_VEL
LIN {X 0,Y 608.483,Z 745.814,A -85,B 0,C 180,E1 -414.369,E2 -414.369} C_VEL
LIN {X 0,Y 608.522,Z 753.592,A -85,B 0,C 180,E1 -416.729,E2 -416.729} C_VEL
LIN {X 0,Y 608.532,Z 762.859,A -85,B 0,C 180,E1 -419.458,E2 -419.458} C_VEL
LIN {X 0,Y 608.501,Z 772.127,A -85,B 0,C 180,E1 -422.111,E2 -422.111} C_VEL
LIN {X 0,Y 608.478,Z 781.394,A -85,B 0,C 180,E1 -424.7,E2 -424.7} C_VEL
LIN {X 0,Y 608.481,Z 791.985,A -85,B 0,C 180,E1 -427.595,E2 -427.595} C_VEL
LIN {X 0,Y 608.46,Z 802.577,A -85,B 0,C 180,E1 -430.43,E2 -430.43} C_VEL
LIN {X 0,Y 608.442,Z 813.168,A -85,B 0,C 180,E1 -433.216,E2 -433.216} C_VEL
LIN {X 0,Y 608.44,Z 823.888,A -85,B 0,C 180,E1 -435.995,E2 -435.995} C_VEL
LIN {X 0,Y 608.435,Z 832.53,A -85,B 0,C 180,E1 -438.211,E2 -438.211} C_VEL
LIN {X 0,Y 608.541,Z 847.695,A -85,B 0,C 180,E1 -438.53,E2 -438.53} C_VEL
LIN {X 0,Y 608.501,Z 859.358,A -85,B 0,C 180,E1 -438.897,E2 -438.897} C_VEL
LIN {X 0,Y 608.504,Z 871.92,A -85,B 0,C 180,E1 -439.435,E2 -439.435} C_VEL
LIN {X 0,Y 608.473,Z 882.578,A -85,B 0,C 180,E1 -440.023,E2 -440.023} C_VEL
LIN {X 0,Y 608.483,Z 893.473,A -85,B 0,C 180,E1 -440.778,E2 -440.778} C_VEL
LIN {X 0,Y 608.475,Z 904.111,A -85,B 0,C 180,E1 -441.699,E2 -441.699} C_VEL
LIN {X 0,Y 608.471,Z 911.96,A -85,B 0,C 180,E1 -442.534,E2 -442.534} C_VEL
LIN {X 0,Y 608.461,Z 919.287,A -85,B 0,C 180,E1 -443.485,E2 -443.485} C_VEL
LIN {X 0,Y 608.45,Z 924.866,A -85,B 0,C 180,E1 -444.366,E2 -444.366} C_VEL
LIN {X 0,Y 608.432,Z 929.95,A -85,B 0,C 180,E1 -445.362,E2 -445.362} C_VEL
LIN {X 0,Y 608.449,Z 933.896,A -85,B 0,C 180,E1 -446.358,E2 -446.358} C_VEL
LIN {X 0,Y 608.425,Z 936.809,A -85,B 0,C 180,E1 -447.352,E2 -447.352} C_VEL
LIN {X 0,Y 608.441,Z 938.201,A -85,B 0,C 180,E1 -448.014,E2 -448.014} C_VEL
LIN {X 0,Y 608.438,Z 939.783,A -85,B 0,C 180,E1 -449.338,E2 -449.338} C_VEL
LIN {X 0,Y 608.434,Z 940,A -85,B 0,C 180,E1 -450,E2 -450} C_VEL
LIN {X 0,Y 608.448,Z 939.184,A -85,B 0,C 180,E1 -451.324,E2 -451.324} C_VEL
LIN {X 0,Y 608.441,Z 938.201,A -85,B 0,C 180,E1 -451.986,E2 -451.986} C_VEL
LIN {X 0,Y 608.425,Z 936.809,A -85,B 0,C 180,E1 -452.648,E2 -452.648} C_VEL
LIN {X 0,Y 608.449,Z 933.896,A -85,B 0,C 180,E1 -453.642,E2 -453.642} C_VEL
LIN {X 0,Y 608.432,Z 929.95,A -85,B 0,C 180,E1 -454.638,E2 -454.638} C_VEL
LIN {X 0,Y 608.437,Z 923.876,A -85,B 0,C 180,E1 -455.801,E2 -455.801} C_VEL
LIN {X 0,Y 608.462,Z 917.235,A -85,B 0,C 180,E1 -456.799,E2 -456.799} C_VEL
LIN {X 0,Y 608.456,Z 908.989,A -85,B 0,C 180,E1 -457.8,E2 -457.8} C_VEL
LIN {X 0,Y 608.472,Z 900.536,A -85,B 0,C 180,E1 -458.636,E2 -458.636} C_VEL
LIN {X 0,Y 608.48,Z 890.09,A -85,B 0,C 180,E1 -459.473,E2 -459.473} C_VEL
LIN {X 0,Y 608.482,Z 879.754,A -85,B 0,C 180,E1 -460.145,E2 -460.145} C_VEL
LIN {X 0,Y 608.497,Z 868.306,A -85,B 0,C 180,E1 -460.739,E2 -460.739} C_VEL
LIN {X 0,Y 608.533,Z 855.951,A -85,B 0,C 180,E1 -461.223,E2 -461.223} C_VEL
LIN {X 0,Y 608.54,Z 842.436,A -85,B 0,C 180,E1 -461.597,E2 -461.597} C_VEL
LIN {X 0,Y 608.435,Z 832.53,A -85,B 0,C 180,E1 -461.789,E2 -461.789} C_VEL
LIN {X 0,Y 608.446,Z 822.435,A -85,B 0,C 180,E1 -464.379,E2 -464.379} C_VEL
LIN {X 0,Y 608.439,Z 811.844,A -85,B 0,C 180,E1 -467.13,E2 -467.13} C_VEL
LIN {X 0,Y 608.46,Z 802.577,A -85,B 0,C 180,E1 -469.57,E2 -469.57} C_VEL
LIN {X 0,Y 608.463,Z 791.725,A -85,B 0,C 180,E1 -472.476,E2 -472.476} C_VEL
LIN {X 0,Y 608.478,Z 781.394,A -85,B 0,C 180,E1 -475.3,E2 -475.3} C_VEL
LIN {X 0,Y 608.501,Z 772.127,A -85,B 0,C 180,E1 -477.889,E2 -477.889} C_VEL
LIN {X 0,Y 608.532,Z 762.859,A -85,B 0,C 180,E1 -480.542,E2 -480.542} C_VEL
LIN {X 0,Y 608.522,Z 753.592,A -85,B 0,C 180,E1 -483.271,E2 -483.271} C_VEL
LIN {X 0,Y 608.478,Z 745.689,A -85,B 0,C 180,E1 -485.682,E2 -485.682} C_VEL
LIN {X 0,Y 608.47,Z 745.686,A -85,B 0,C 180,E1 -488.24,E2 -488.24} C_VEL
LIN {X 0,Y 608.457,Z 745.693,A -85,B 0,C 180,E1 -491.341,E2 -491.341} C_VEL
LIN {X 0,Y 608.462,Z 745.687,A -85,B 0,C 180,E1 -494.264,E2 -494.264} C_VEL
LIN {X 0,Y 608.454,Z 745.698,A -85,B 0,C 180,E1 -497.04,E2 -497.04} C_VEL
LIN {X 0,Y 608.457,Z 745.688,A -85,B 0,C 180,E1 -499.697,E2 -499.697} C_VEL
LIN {X 0,Y 608.483,Z 745.693,A -85,B 0,C 180,E1 -502.84,E2 -502.84} C_VEL
LIN {X 0,Y 608.434,Z 745.918,A -85,B 0,C 180,E1 -505.097,E2 -505.097} C_VEL
LIN {X 0,Y 608.417,Z 748.801,A -85,B 0,C 180,E1 -507.485,E2 -507.485} C_VEL
LIN {X 0,Y 608.428,Z 751.966,A -85,B 0,C 180,E1 -510.036,E2 -510.036} C_VEL
LIN {X 0,Y 608.431,Z 755.492,A -85,B 0,C 180,E1 -512.802,E2 -512.802} C_VEL
LIN {X 0,Y 608.419,Z 758.92,A -85,B 0,C 180,E1 -515.427,E2 -515.427} C_VEL
LIN {X 0,Y 608.403,Z 762.763,A -85,B 0,C 180,E1 -518.305,E2 -518.305} C_VEL
LIN {X 0,Y 608.438,Z 766.607,A -85,B 0,C 180,E1 -521.129,E2 -521.129} C_VEL
LIN {X 0,Y 608.414,Z 770.45,A -85,B 0,C 180,E1 -523.904,E2 -523.904} C_VEL
LIN {X 0,Y 608.428,Z 774.293,A -85,B 0,C 180,E1 -526.642,E2 -526.642} C_VEL
LIN {X 0,Y 608.424,Z 776.665,A -85,B 0,C 180,E1 -528.316,E2 -528.316} C_VEL
LIN {X 0,Y 608.534,Z 792.48,A -85,B 0,C 180,E1 -528.709,E2 -528.709} C_VEL
LIN {X 0,Y 608.519,Z 804.774,A -85,B 0,C 180,E1 -529.155,E2 -529.155} C_VEL
LIN {X 0,Y 608.487,Z 817.489,A -85,B 0,C 180,E1 -529.771,E2 -529.771} C_VEL
LIN {X 0,Y 608.486,Z 828.296,A -85,B 0,C 180,E1 -530.442,E2 -530.442} C_VEL
LIN {X 0,Y 608.477,Z 838.07,A -85,B 0,C 180,E1 -531.196,E2 -531.196} C_VEL
LIN {X 0,Y 608.46,Z 846.969,A -85,B 0,C 180,E1 -532.032,E2 -532.032} C_VEL
LIN {X 0,Y 608.465,Z 855.658,A -85,B 0,C 180,E1 -533.033,E2 -533.033} C_VEL
LIN {X 0,Y 608.439,Z 862.589,A -85,B 0,C 180,E1 -534.032,E2 -534.032} C_VEL
LIN {X 0,Y 608.436,Z 868.143,A -85,B 0,C 180,E1 -535.029,E2 -535.029} C_VEL
LIN {X 0,Y 608.434,Z 872.506,A -85,B 0,C 180,E1 -536.025,E2 -536.025} C_VEL
LIN {X 0,Y 608.425,Z 874.81,A -85,B 0,C 180,E1 -536.688,E2 -536.688} C_VEL
LIN {X 0,Y 608.427,Z 876.689,A -85,B 0,C 180,E1 -537.351,E2 -537.351} C_VEL
LIN {X 0,Y 608.442,Z 878.126,A -85,B 0,C 180,E1 -538.014,E2 -538.014} C_VEL
LIN {X 0,Y 608.44,Z 879.751,A -85,B 0,C 180,E1 -539.337,E2 -539.337} C_VEL
LIN {X 0,Y 608.434,Z 879.995,A -85,B 0,C 180,E1 -539.999,E2 -539.999} C_VEL
LIN {X 0,Y 608.438,Z 879.816,A -85,B 0,C 180,E1 -540.661,E2 -540.661} C_VEL
LIN {X 0,Y 608.442,Z 878.277,A -85,B 0,C 180,E1 -541.985,E2 -541.985} C_VEL
LIN {X 0,Y 608.426,Z 876.92,A -85,B 0,C 180,E1 -542.648,E2 -542.648} C_VEL
LIN {X 0,Y 608.45,Z 874.044,A -85,B 0,C 180,E1 -543.642,E2 -543.642} C_VEL
LIN {X 0,Y 608.433,Z 870.146,A -85,B 0,C 180,E1 -544.637,E2 -544.637} C_VEL
LIN {X 0,Y 608.449,Z 865.116,A -85,B 0,C 180,E1 -545.634,E2 -545.634} C_VEL
LIN {X 0,Y 608.441,Z 858.8,A -85,B 0,C 180,E1 -546.632,E2 -546.632} C_VEL
LIN {X 0,Y 608.475,Z 850.885,A -85,B 0,C 180,E1 -547.632,E2 -547.632} C_VEL
LIN {X 0,Y 608.472,Z 841.044,A -85,B 0,C 180,E1 -548.635,E2 -548.635} C_VEL
LIN {X 0,Y 608.477,Z 838.936,A -85,B 0,C 180,E1 -548.819,E2 -548.819} C_VEL
LIN {X 0,Y 607.812,Z 834.601,A -85,B 0,C 180,E1 -549.19,E2 -549.19} C_VEL
LIN {X 0,Y 604.974,Z 827.351,A -85,B 0,C 180,E1 -549.769,E2 -549.769} C_VEL
LIN {X 0,Y 602.148,Z 819.707,A -85,B 0,C 180,E1 -550.301,E2 -550.301} C_VEL
LIN {X 0,Y 601.505,Z 814.643,A -85,B 0,C 180,E1 -550.595,E2 -550.595} C_VEL
LIN {X 0,Y 601.51,Z 802.407,A -85,B 0,C 180,E1 -551.163,E2 -551.163} C_VEL
LIN {X 0,Y 601.552,Z 789.326,A -85,B 0,C 180,E1 -551.605,E2 -551.605} C_VEL
LIN {X 0,Y 601.396,Z 777.249,A -85,B 0,C 180,E1 -551.885,E2 -551.885} C_VEL
LIN {X 0,Y 601.345,Z 776.644,A -85,B 0,C 180,E1 -551.929,E2 -551.929} C_VEL
LIN {X 0,Y 601.321,Z 773.46,A -85,B 0,C 180,E1 -554.207,E2 -554.207} C_VEL
LIN {X 0,Y 601.328,Z 769.615,A -85,B 0,C 180,E1 -556.988,E2 -556.988} C_VEL
LIN {X 0,Y 601.317,Z 765.77,A -85,B 0,C 180,E1 -559.812,E2 -559.812} C_VEL
LIN {X 0,Y 601.332,Z 762.057,A -85,B 0,C 180,E1 -562.585,E2 -562.585} C_VEL
LIN {X 0,Y 601.342,Z 759.04,A -85,B 0,C 180,E1 -564.88,E2 -564.88} C_VEL
LIN {X 0,Y 601.341,Z 755.859,A -85,B 0,C 180,E1 -567.348,E2 -567.348} C_VEL
LIN {X 0,Y 601.348,Z 752.31,A -85,B 0,C 180,E1 -570.167,E2 -570.167} C_VEL
LIN {X 0,Y 601.365,Z 749.198,A -85,B 0,C 180,E1 -572.707,E2 -572.707} C_VEL
LIN {X 0,Y 601.371,Z 746.58,A -85,B 0,C 180,E1 -575.108,E2 -575.108} C_VEL
LIN {X 0,Y 601.431,Z 746.569,A -85,B 0,C 180,E1 -577.418,E2 -577.418} C_VEL
LIN {X 0,Y 601.396,Z 746.567,A -85,B 0,C 180,E1 -579.995,E2 -579.995} C_VEL
LIN {X 0,Y 601.407,Z 746.566,A -85,B 0,C 180,E1 -582.669,E2 -582.669} C_VEL
LIN {X 0,Y 601.421,Z 746.572,A -85,B 0,C 180,E1 -585.481,E2 -585.481} C_VEL
LIN {X 0,Y 601.411,Z 746.564,A -85,B 0,C 180,E1 -588.407,E2 -588.407} C_VEL
LIN {X 0,Y 601.41,Z 746.566,A -85,B 0,C 180,E1 -590.873,E2 -590.873} C_VEL
LIN {X 0,Y 601.403,Z 746.575,A -85,B 0,C 180,E1 -593.417,E2 -593.417} C_VEL
LIN {X 0,Y 601.396,Z 746.568,A -85,B 0,C 180,E1 -596.068,E2 -596.068} C_VEL
LIN {X 0,Y 601.406,Z 746.565,A -85,B 0,C 180,E1 -598.546,E2 -598.546} C_VEL
LIN {X 0,Y 601.439,Z 746.567,A -85,B 0,C 180,E1 -601.373,E2 -601.373} C_VEL
LIN {X 0,Y 601.381,Z 746.571,A -85,B 0,C 180,E1 -604.137,E2 -604.137} C_VEL
LIN {X 0,Y 601.368,Z 746.569,A -85,B 0,C 180,E1 -606.587,E2 -606.587} C_VEL
LIN {X 0,Y 601.426,Z 746.569,A -85,B 0,C 180,E1 -609.478,E2 -609.478} C_VEL
LIN {X 0,Y 601.363,Z 746.572,A -85,B 0,C 180,E1 -612.311,E2 -612.311} C_VEL
LIN {X 0,Y 601.375,Z 746.57,A -85,B 0,C 180,E1 -614.408,E2 -614.408} C_VEL
LIN {X 0,Y 601.373,Z 746.57,A -85,B 0,C 180,E1 -616.483,E2 -616.483} C_VEL
LIN {X 0,Y 601.37,Z 746.57,A -85,B 0,C 180,E1 -619.223,E2 -619.223} C_VEL
LIN {X 0,Y 601.421,Z 746.574,A -85,B 0,C 180,E1 -621.939,E2 -621.939} C_VEL
LIN {X 0,Y 601.374,Z 746.57,A -85,B 0,C 180,E1 -624.635,E2 -624.635} C_VEL
LIN {X 0,Y 601.388,Z 746.568,A -85,B 0,C 180,E1 -627.321,E2 -627.321} C_VEL
LIN {X 0,Y 601.434,Z 746.572,A -85,B 0,C 180,E1 -630,E2 -630} C_VEL
LIN {X 0,Y 601.387,Z 746.569,A -85,B 0,C 180,E1 -632.679,E2 -632.679} C_VEL
LIN {X 0,Y 601.365,Z 746.57,A -85,B 0,C 180,E1 -635.365,E2 -635.365} C_VEL
LIN {X 0,Y 601.392,Z 746.576,A -85,B 0,C 180,E1 -638.061,E2 -638.061} C_VEL
LIN {X 0,Y 601.365,Z 746.572,A -85,B 0,C 180,E1 -640.777,E2 -640.777} C_VEL
LIN {X 0,Y 601.362,Z 746.571,A -85,B 0,C 180,E1 -643.517,E2 -643.517} C_VEL
LIN {X 0,Y 601.426,Z 746.573,A -85,B 0,C 180,E1 -646.287,E2 -646.287} C_VEL
LIN {X 0,Y 601.394,Z 746.567,A -85,B 0,C 180,E1 -649.1,E2 -649.1} C_VEL
LIN {X 0,Y 601.377,Z 746.568,A -85,B 0,C 180,E1 -651.241,E2 -651.241} C_VEL
LIN {X 0,Y 601.431,Z 746.568,A -85,B 0,C 180,E1 -654.142,E2 -654.142} C_VEL
LIN {X 0,Y 601.408,Z 746.566,A -85,B 0,C 180,E1 -657.113,E2 -657.113} C_VEL
LIN {X 0,Y 601.389,Z 746.567,A -85,B 0,C 180,E1 -659.395,E2 -659.395} C_VEL
LIN {X 0,Y 601.383,Z 746.568,A -85,B 0,C 180,E1 -661.728,E2 -661.728} C_VEL
LIN {X 0,Y 601.406,Z 746.568,A -85,B 0,C 180,E1 -664.12,E2 -664.12} C_VEL
LIN {X 0,Y 601.427,Z 746.563,A -85,B 0,C 180,E1 -667.383,E2 -667.383} C_VEL
LIN {X 0,Y 601.393,Z 746.568,A -85,B 0,C 180,E1 -669.997,E2 -669.997} C_VEL
LIN {X 0,Y 601.405,Z 746.576,A -85,B 0,C 180,E1 -672.671,E2 -672.671} C_VEL
LIN {X 0,Y 601.393,Z 746.567,A -85,B 0,C 180,E1 -675.48,E2 -675.48} C_VEL
LIN {X 0,Y 601.413,Z 746.568,A -85,B 0,C 180,E1 -678.408,E2 -678.408} C_VEL
LIN {X 0,Y 601.405,Z 746.575,A -85,B 0,C 180,E1 -680.874,E2 -680.874} C_VEL
LIN {X 0,Y 601.403,Z 746.567,A -85,B 0,C 180,E1 -683.418,E2 -683.418} C_VEL
LIN {X 0,Y 601.375,Z 746.579,A -85,B 0,C 180,E1 -685.067,E2 -685.067} C_VEL
LIN {X 0,Y 601.377,Z 749.317,A -85,B 0,C 180,E1 -687.482,E2 -687.482} C_VEL
LIN {X 0,Y 601.349,Z 752.239,A -85,B 0,C 180,E1 -689.865,E2 -689.865} C_VEL
LIN {X 0,Y 601.344,Z 755.743,A -85,B 0,C 180,E1 -692.651,E2 -692.651} C_VEL
LIN {X 0,Y 601.345,Z 758.923,A -85,B 0,C 180,E1 -695.12,E2 -695.12} C_VEL
LIN {X 0,Y 601.339,Z 762.766,A -85,B 0,C 180,E1 -698.039,E2 -698.039} C_VEL
LIN {X 0,Y 601.319,Z 765.648,A -85,B 0,C 180,E1 -700.188,E2 -700.188} C_VEL
LIN {X 0,Y 601.33,Z 769.492,A -85,B 0,C 180,E1 -703.012,E2 -703.012} C_VEL
LIN {X 0,Y 601.349,Z 773.535,A -85,B 0,C 180,E1 -705.937,E2 -705.937} C_VEL
LIN {X 0,Y 601.351,Z 776.668,A -85,B 0,C 180,E1 -708.178,E2 -708.178} C_VEL
LIN {X 0,Y 601.573,Z 786.876,A -85,B 0,C 180,E1 -708.417,E2 -708.417} C_VEL
LIN {X 0,Y 601.519,Z 800.039,A -85,B 0,C 180,E1 -708.837,E2 -708.837} C_VEL
LIN {X 0,Y 601.506,Z 812.76,A -85,B 0,C 180,E1 -709.397,E2 -709.397} C_VEL
LIN {X 0,Y 601.488,Z 824.532,A -85,B 0,C 180,E1 -710.077,E2 -710.077} C_VEL
LIN {X 0,Y 601.438,Z 836.101,A -85,B 0,C 180,E1 -710.924,E2 -710.924} C_VEL
LIN {X 0,Y 601.411,Z 845.359,A -85,B 0,C 180,E1 -711.77,E2 -711.77} C_VEL
LIN {X 0,Y 601.388,Z 854.33,A -85,B 0,C 180,E1 -712.784,E2 -712.784} C_VEL
LIN {X 0,Y 601.376,Z 861.464,A -85,B 0,C 180,E1 -713.781,E2 -713.781} C_VEL
LIN {X 0,Y 601.372,Z 866.435,A -85,B 0,C 180,E1 -714.636,E2 -714.636} C_VEL
LIN {X 0,Y 601.353,Z 871.18,A -85,B 0,C 180,E1 -715.644,E2 -715.644} C_VEL
LIN {X 0,Y 601.345,Z 874.814,A -85,B 0,C 180,E1 -716.651,E2 -716.651} C_VEL
LIN {X 0,Y 601.324,Z 876.695,A -85,B 0,C 180,E1 -717.321,E2 -717.321} C_VEL
LIN {X 0,Y 601.341,Z 878.129,A -85,B 0,C 180,E1 -717.991,E2 -717.991} C_VEL
LIN {X 0,Y 601.339,Z 879.753,A -85,B 0,C 180,E1 -719.331,E2 -719.331} C_VEL
LIN {X 0,Y 601.335,Z 879.996,A -85,B 0,C 180,E1 -720.001,E2 -720.001} C_VEL
LIN {X 0,Y 601.339,Z 879.815,A -85,B 0,C 180,E1 -720.67,E2 -720.67} C_VEL
LIN {X 0,Y 601.34,Z 878.275,A -85,B 0,C 180,E1 -722.01,E2 -722.01} C_VEL
LIN {X 0,Y 601.326,Z 876.909,A -85,B 0,C 180,E1 -722.68,E2 -722.68} C_VEL
LIN {X 0,Y 601.368,Z 874.033,A -85,B 0,C 180,E1 -723.686,E2 -723.686} C_VEL
LIN {X 0,Y 601.337,Z 870.132,A -85,B 0,C 180,E1 -724.693,E2 -724.693} C_VEL
LIN {X 0,Y 601.373,Z 865.102,A -85,B 0,C 180,E1 -725.702,E2 -725.702} C_VEL
LIN {X 0,Y 601.383,Z 858.786,A -85,B 0,C 180,E1 -726.712,E2 -726.712} C_VEL
LIN {X 0,Y 601.396,Z 850.869,A -85,B 0,C 180,E1 -727.724,E2 -727.724} C_VEL
LIN {X 0,Y 601.422,Z 842.802,A -85,B 0,C 180,E1 -728.569,E2 -728.569} C_VEL
LIN {X 0,Y 601.454,Z 832.964,A -85,B 0,C 180,E1 -729.416,E2 -729.416} C_VEL
LIN {X 0,Y 601.463,Z 821.907,A -85,B 0,C 180,E1 -730.18,E2 -730.18} C_VEL
LIN {X 0,Y 601.52,Z 809.842,A -85,B 0,C 180,E1 -730.836,E2 -730.836} C_VEL
LIN {X 0,Y 601.556,Z 797.697,A -85,B 0,C 180,E1 -731.341,E2 -731.341} C_VEL
LIN {X 0,Y 601.603,Z 785.232,A -85,B 0,C 180,E1 -731.712,E2 -731.712} C_VEL
LIN {X 0,Y 601.333,Z 776.673,A -85,B 0,C 180,E1 -731.909,E2 -731.909} C_VEL
LIN {X 0,Y 601.319,Z 773.458,A -85,B 0,C 180,E1 -734.208,E2 -734.208} C_VEL
LIN {X 0,Y 601.337,Z 769.613,A -85,B 0,C 180,E1 -736.989,E2 -736.989} C_VEL
LIN {X 0,Y 601.31,Z 765.768,A -85,B 0,C 180,E1 -739.813,E2 -739.813} C_VEL
LIN {X 0,Y 601.337,Z 762.884,A -85,B 0,C 180,E1 -741.963,E2 -741.963} C_VEL
LIN {X 0,Y 601.341,Z 759.038,A -85,B 0,C 180,E1 -744.882,E2 -744.882} C_VEL
LIN {X 0,Y 601.345,Z 755.858,A -85,B 0,C 180,E1 -747.349,E2 -747.349} C_VEL
LIN {X 0,Y 601.345,Z 752.308,A -85,B 0,C 180,E1 -750.169,E2 -750.169} C_VEL
LIN {X 0,Y 601.352,Z 749.202,A -85,B 0,C 180,E1 -752.705,E2 -752.705} C_VEL
LIN {X 0,Y 601.38,Z 746.579,A -85,B 0,C 180,E1 -755.109,E2 -755.109} C_VEL
LIN {X 0,Y 601.438,Z 746.567,A -85,B 0,C 180,E1 -757.419,E2 -757.419} C_VEL
LIN {X 0,Y 601.415,Z 746.564,A -85,B 0,C 180,E1 -759.995,E2 -759.995} C_VEL
LIN {X 0,Y 601.391,Z 746.571,A -85,B 0,C 180,E1 -762.673,E2 -762.673} C_VEL
LIN {X 0,Y 601.431,Z 746.565,A -85,B 0,C 180,E1 -765.482,E2 -765.482} C_VEL
LIN {X 0,Y 601.423,Z 746.565,A -85,B 0,C 180,E1 -768.407,E2 -768.407} C_VEL
LIN {X 0,Y 601.436,Z 746.564,A -85,B 0,C 180,E1 -771.529,E2 -771.529} C_VEL
LIN {X 0,Y 601.464,Z 746.681,A -85,B 0,C 180,E1 -774.16,E2 -774.16} C_VEL
LIN {X 0,Y 601.588,Z 752.764,A -85,B 0,C 180,E1 -776.043,E2 -776.043} C_VEL
LIN {X 0,Y 601.57,Z 761.02,A -85,B 0,C 180,E1 -778.523,E2 -778.523} C_VEL
LIN {X 0,Y 601.5,Z 770.803,A -85,B 0,C 180,E1 -781.377,E2 -781.377} C_VEL
LIN {X 0,Y 601.482,Z 780.451,A -85,B 0,C 180,E1 -784.12,E2 -784.12} C_VEL
LIN {X 0,Y 601.468,Z 789.338,A -85,B 0,C 180,E1 -786.592,E2 -786.592} C_VEL
LIN {X 0,Y 601.432,Z 799.929,A -85,B 0,C 180,E1 -789.478,E2 -789.478} C_VEL
LIN {X 0,Y 601.403,Z 810.52,A -85,B 0,C 180,E1 -792.312,E2 -792.312} C_VEL
LIN {X 0,Y 601.364,Z 821.111,A -85,B 0,C 180,E1 -795.101,E2 -795.101} C_VEL
LIN {X 0,Y 601.364,Z 831.703,A -85,B 0,C 180,E1 -797.856,E2 -797.856} C_VEL
LIN {X 0,Y 601.381,Z 832.53,A -85,B 0,C 180,E1 -798.071,E2 -798.071} C_VEL
LIN {X 0,Y 601.616,Z 846.931,A -85,B 0,C 180,E1 -798.375,E2 -798.375} C_VEL
LIN {X 0,Y 601.544,Z 859.183,A -85,B 0,C 180,E1 -798.76,E2 -798.76} C_VEL
LIN {X 0,Y 601.508,Z 871.921,A -85,B 0,C 180,E1 -799.311,E2 -799.311} C_VEL
LIN {X 0,Y 601.466,Z 882.579,A -85,B 0,C 180,E1 -799.905,E2 -799.905} C_VEL
LIN {X 0,Y 601.449,Z 893.474,A -85,B 0,C 180,E1 -800.669,E2 -800.669} C_VEL
LIN {X 0,Y 601.429,Z 904.111,A -85,B 0,C 180,E1 -801.601,E2 -801.601} C_VEL
LIN {X 0,Y 601.418,Z 911.96,A -85,B 0,C 180,E1 -802.446,E2 -802.446} C_VEL
LIN {X 0,Y 601.37,Z 919.225,A -85,B 0,C 180,E1 -803.398,E2 -803.398} C_VEL
LIN {X 0,Y 601.372,Z 924.866,A -85,B 0,C 180,E1 -804.299,E2 -804.299} C_VEL
LIN {X 0,Y 601.336,Z 929.95,A -85,B 0,C 180,E1 -805.307,E2 -805.307} C_VEL
LIN {X 0,Y 601.367,Z 933.896,A -85,B 0,C 180,E1 -806.315,E2 -806.315} C_VEL
LIN {X 0,Y 601.325,Z 936.809,A -85,B 0,C 180,E1 -807.32,E2 -807.32} C_VEL
LIN {X 0,Y 601.34,Z 938.201,A -85,B 0,C 180,E1 -807.991,E2 -807.991} C_VEL
LIN {X 0,Y 601.339,Z 939.784,A -85,B 0,C 180,E1 -809.33,E2 -809.33} C_VEL
LIN {X 0,Y 601.335,Z 940,A -85,B 0,C 180,E1 -810,E2 -810} C_VEL
LIN {X 0,Y 601.348,Z 939.184,A -85,B 0,C 180,E1 -811.339,E2 -811.339} C_VEL
LIN {X 0,Y 601.34,Z 938.202,A -85,B 0,C 180,E1 -812.009,E2 -812.009} C_VEL
LIN {X 0,Y 601.325,Z 936.809,A -85,B 0,C 180,E1 -812.68,E2 -812.68} C_VEL
LIN {X 0,Y 601.367,Z 933.896,A -85,B 0,C 180,E1 -813.685,E2 -813.685} C_VEL
LIN {X 0,Y 601.336,Z 929.95,A -85,B 0,C 180,E1 -814.693,E2 -814.693} C_VEL
LIN {X 0,Y 601.372,Z 923.877,A -85,B 0,C 180,E1 -815.869,E2 -815.869} C_VEL
LIN {X 0,Y 601.382,Z 917.235,A -85,B 0,C 180,E1 -816.88,E2 -816.88} C_VEL
LIN {X 0,Y 601.4,Z 908.989,A -85,B 0,C 180,E1 -817.892,E2 -817.892} C_VEL
LIN {X 0,Y 601.436,Z 900.536,A -85,B 0,C 180,E1 -818.738,E2 -818.738} C_VEL
LIN {X 0,Y 601.446,Z 890.091,A -85,B 0,C 180,E1 -819.585,E2 -819.585} C_VEL
LIN {X 0,Y 601.479,Z 879.755,A -85,B 0,C 180,E1 -820.264,E2 -820.264} C_VEL
LIN {X 0,Y 601.51,Z 867.922,A -85,B 0,C 180,E1 -820.882,E2 -820.882} C_VEL
LIN {X 0,Y 601.562,Z 855.275,A -85,B 0,C 180,E1 -821.377,E2 -821.377} C_VEL
LIN {X 0,Y 601.594,Z 842.436,A -85,B 0,C 180,E1 -821.733,E2 -821.733} C_VEL
LIN {X 0,Y 601.381,Z 832.53,A -85,B 0,C 180,E1 -821.929,E2 -821.929} C_VEL
LIN {X 0,Y 601.389,Z 822.435,A -85,B 0,C 180,E1 -824.552,E2 -824.552} C_VEL
LIN {X 0,Y 601.39,Z 811.844,A -85,B 0,C 180,E1 -827.338,E2 -827.338} C_VEL
LIN {X 0,Y 601.423,Z 801.253,A -85,B 0,C 180,E1 -830.165,E2 -830.165} C_VEL
LIN {X 0,Y 601.434,Z 791.985,A -85,B 0,C 180,E1 -832.682,E2 -832.682} C_VEL
LIN {X 0,Y 601.462,Z 782.718,A -85,B 0,C 180,E1 -835.246,E2 -835.246} C_VEL
LIN {X 0,Y 601.508,Z 773.451,A -85,B 0,C 180,E1 -837.863,E2 -837.863} C_VEL
LIN {X 0,Y 601.563,Z 764.185,A -85,B 0,C 180,E1 -840.544,E2 -840.544} C_VEL
LIN {X 0,Y 601.581,Z 754.916,A -85,B 0,C 180,E1 -843.304,E2 -843.304} C_VEL
LIN {X 0,Y 601.62,Z 748.923,A -85,B 0,C 180,E1 -845.142,E2 -845.142} C_VEL
LIN {X 0,Y 601.437,Z 746.568,A -85,B 0,C 180,E1 -845.931,E2 -845.931} C_VEL
LIN {X 0,Y 601.437,Z 746.564,A -85,B 0,C 180,E1 -848.471,E2 -848.471} C_VEL
LIN {X 0,Y 601.425,Z 746.566,A -85,B 0,C 180,E1 -851.593,E2 -851.593} C_VEL
LIN {X 0,Y 601.43,Z 746.566,A -85,B 0,C 180,E1 -854.535,E2 -854.535} C_VEL
LIN {X 0,Y 601.39,Z 746.573,A -85,B 0,C 180,E1 -857.327,E2 -857.327} C_VEL
LIN {X 0,Y 601.407,Z 746.566,A -85,B 0,C 180,E1 -860.004,E2 -860.004} C_VEL
LIN {X 0,Y 601.44,Z 746.567,A -85,B 0,C 180,E1 -862.618,E2 -862.618} C_VEL
LIN {X 0,Y 601.381,Z 746.579,A -85,B 0,C 180,E1 -865.065,E2 -865.065} C_VEL
LIN {X 0,Y 601.356,Z 749.315,A -85,B 0,C 180,E1 -867.479,E2 -867.479} C_VEL
LIN {X 0,Y 601.346,Z 752.239,A -85,B 0,C 180,E1 -869.866,E2 -869.866} C_VEL
LIN {X 0,Y 601.345,Z 755.743,A -85,B 0,C 180,E1 -872.651,E2 -872.651} C_VEL
LIN {X 0,Y 601.342,Z 759.717,A -85,B 0,C 180,E1 -875.728,E2 -875.728} C_VEL
LIN {X 0,Y 601.331,Z 762.764,A -85,B 0,C 180,E1 -878.037,E2 -878.037} C_VEL
LIN {X 0,Y 601.308,Z 765.646,A -85,B 0,C 180,E1 -880.187,E2 -880.187} C_VEL
LIN {X 0,Y 601.338,Z 769.49,A -85,B 0,C 180,E1 -883.011,E2 -883.011} C_VEL
LIN {X 0,Y 601.324,Z 773.549,A -85,B 0,C 180,E1 -885.947,E2 -885.947} C_VEL
LIN {X 0,Y 601.332,Z 776.666,A -85,B 0,C 180,E1 -888.176,E2 -888.176} C_VEL
LIN {X 0,Y 601.592,Z 781.398,A -85,B 0,C 180,E1 -888.288,E2 -888.288} C_VEL
LIN {X 0,Y 601.568,Z 793.832,A -85,B 0,C 180,E1 -888.621,E2 -888.621} C_VEL
LIN {X 0,Y 601.548,Z 805.809,A -85,B 0,C 180,E1 -889.072,E2 -889.072} C_VEL
LIN {X 0,Y 601.492,Z 817.501,A -85,B 0,C 180,E1 -889.65,E2 -889.65} C_VEL
LIN {X 0,Y 601.457,Z 828.303,A -85,B 0,C 180,E1 -890.33,E2 -890.33} C_VEL
LIN {X 0,Y 601.435,Z 838.077,A -85,B 0,C 180,E1 -891.092,E2 -891.092} C_VEL
LIN {X 0,Y 601.407,Z 846.975,A -85,B 0,C 180,E1 -891.938,E2 -891.938} C_VEL
LIN {X 0,Y 601.385,Z 855.662,A -85,B 0,C 180,E1 -892.951,E2 -892.951} C_VEL
LIN {X 0,Y 601.361,Z 862.592,A -85,B 0,C 180,E1 -893.962,E2 -893.962} C_VEL
LIN {X 0,Y 601.345,Z 868.146,A -85,B 0,C 180,E1 -894.971,E2 -894.971} C_VEL
LIN {X 0,Y 601.346,Z 872.508,A -85,B 0,C 180,E1 -895.978,E2 -895.978} C_VEL
LIN {X 0,Y 601.344,Z 874.812,A -85,B 0,C 180,E1 -896.649,E2 -896.649} C_VEL
LIN {X 0,Y 601.327,Z 876.691,A -85,B 0,C 180,E1 -897.32,E2 -897.32} C_VEL
LIN {X 0,Y 601.341,Z 878.126,A -85,B 0,C 180,E1 -897.99,E2 -897.99} C_VEL
LIN {X 0,Y 601.34,Z 879.752,A -85,B 0,C 180,E1 -899.33,E2 -899.33} C_VEL
LIN {X 0,Y 601.335,Z 879.995,A -85,B 0,C 180,E1 -899.999,E2 -899.999} C_VEL
LIN {X 0,Y 601.339,Z 879.815,A -85,B 0,C 180,E1 -900.669,E2 -900.669} C_VEL
LIN {X 0,Y 601.341,Z 878.277,A -85,B 0,C 180,E1 -902.009,E2 -902.009} C_VEL
LIN {X 0,Y 601.326,Z 876.918,A -85,B 0,C 180,E1 -902.679,E2 -902.679} C_VEL
LIN {X 0,Y 601.369,Z 874.042,A -85,B 0,C 180,E1 -903.685,E2 -903.685} C_VEL
LIN {X 0,Y 601.337,Z 870.144,A -85,B 0,C 180,E1 -904.692,E2 -904.692} C_VEL
LIN {X 0,Y 601.373,Z 865.113,A -85,B 0,C 180,E1 -905.7,E2 -905.7} C_VEL
LIN {X 0,Y 601.382,Z 858.796,A -85,B 0,C 180,E1 -906.71,E2 -906.71} C_VEL
LIN {X 0,Y 601.396,Z 850.88,A -85,B 0,C 180,E1 -907.723,E2 -907.723} C_VEL
LIN {X 0,Y 601.436,Z 841.038,A -85,B 0,C 180,E1 -908.737,E2 -908.737} C_VEL
LIN {X 0,Y 601.451,Z 830.718,A -85,B 0,C 180,E1 -909.584,E2 -909.584} C_VEL
LIN {X 0,Y 601.485,Z 819.103,A -85,B 0,C 180,E1 -910.348,E2 -910.348} C_VEL
LIN {X 0,Y 601.505,Z 814.643,A -85,B 0,C 180,E1 -910.595,E2 -910.595} C_VEL
LIN {X 0,Y 600.874,Z 809.519,A -85,B 0,C 180,E1 -910.869,E2 -910.869} C_VEL
LIN {X 0,Y 598.098,Z 801.069,A -85,B 0,C 180,E1 -911.288,E2 -911.288} C_VEL
LIN {X 0,Y 595.304,Z 792.324,A -85,B 0,C 180,E1 -911.643,E2 -911.643} C_VEL
LIN {X 0,Y 594.638,Z 786.742,A -85,B 0,C 180,E1 -911.814,E2 -911.814} C_VEL
LIN {X 0,Y 594.455,Z 778.219,A -85,B 0,C 180,E1 -912.007,E2 -912.007} C_VEL
LIN {X 0,Y 594.251,Z 776.644,A -85,B 0,C 180,E1 -912.074,E2 -912.074} C_VEL
LIN {X 0,Y 594.235,Z 773.46,A -85,B 0,C 180,E1 -914.38,E2 -914.38} C_VEL
LIN {X 0,Y 594.231,Z 769.614,A -85,B 0,C 180,E1 -917.197,E2 -917.197} C_VEL
LIN {X 0,Y 594.224,Z 765.769,A -85,B 0,C 180,E1 -920.058,E2 -920.058} C_VEL
LIN {X 0,Y 594.244,Z 762.27,A -85,B 0,C 180,E1 -922.707,E2 -922.707} C_VEL
LIN {X 0,Y 594.253,Z 759.039,A -85,B 0,C 180,E1 -925.198,E2 -925.198} C_VEL
LIN {X 0,Y 594.267,Z 756.107,A -85,B 0,C 180,E1 -927.504,E2 -927.504} C_VEL
LIN {X 0,Y 594.271,Z 752.623,A -85,B 0,C 180,E1 -930.309,E2 -930.309} C_VEL
LIN {X 0,Y 594.293,Z 749.425,A -85,B 0,C 180,E1 -932.954,E2 -932.954} C_VEL
LIN {X 0,Y 594.292,Z 747.541,A -85,B 0,C 180,E1 -934.585,E2 -934.585} C_VEL
LIN {X 0,Y 594.381,Z 747.448,A -85,B 0,C 180,E1 -937.086,E2 -937.086} C_VEL
LIN {X 0,Y 594.352,Z 747.446,A -85,B 0,C 180,E1 -939.771,E2 -939.771} C_VEL
LIN {X 0,Y 594.361,Z 747.443,A -85,B 0,C 180,E1 -942.375,E2 -942.375} C_VEL
LIN {X 0,Y 594.359,Z 747.451,A -85,B 0,C 180,E1 -945.19,E2 -945.19} C_VEL
LIN {X 0,Y 594.367,Z 747.442,A -85,B 0,C 180,E1 -948.152,E2 -948.152} C_VEL
LIN {X 0,Y 594.373,Z 747.447,A -85,B 0,C 180,E1 -951.194,E2 -951.194} C_VEL
LIN {X 0,Y 594.343,Z 747.451,A -85,B 0,C 180,E1 -953.755,E2 -953.755} C_VEL
LIN {X 0,Y 594.348,Z 747.445,A -85,B 0,C 180,E1 -956.237,E2 -956.237} C_VEL
LIN {X 0,Y 594.357,Z 747.443,A -85,B 0,C 180,E1 -958.649,E2 -958.649} C_VEL
LIN {X 0,Y 594.377,Z 747.443,A -85,B 0,C 180,E1 -961.041,E2 -961.041} C_VEL
LIN {X 0,Y 594.346,Z 747.448,A -85,B 0,C 180,E1 -964.054,E2 -964.054} C_VEL
LIN {X 0,Y 594.355,Z 747.445,A -85,B 0,C 180,E1 -966.294,E2 -966.294} C_VEL
LIN {X 0,Y 594.398,Z 747.441,A -85,B 0,C 180,E1 -969.224,E2 -969.224} C_VEL
LIN {X 0,Y 594.329,Z 747.452,A -85,B 0,C 180,E1 -972.094,E2 -972.094} C_VEL
LIN {X 0,Y 594.337,Z 747.449,A -85,B 0,C 180,E1 -974.218,E2 -974.218} C_VEL
LIN {X 0,Y 594.349,Z 747.447,A -85,B 0,C 180,E1 -976.32,E2 -976.32} C_VEL
LIN {X 0,Y 594.352,Z 747.444,A -85,B 0,C 180,E1 -979.094,E2 -979.094} C_VEL
LIN {X 0,Y 594.366,Z 747.452,A -85,B 0,C 180,E1 -981.843,E2 -981.843} C_VEL
LIN {X 0,Y 594.344,Z 747.446,A -85,B 0,C 180,E1 -984.572,E2 -984.572} C_VEL
LIN {X 0,Y 594.356,Z 747.444,A -85,B 0,C 180,E1 -987.289,E2 -987.289} C_VEL
LIN {X 0,Y 594.402,Z 747.448,A -85,B 0,C 180,E1 -990,E2 -990} C_VEL
LIN {X 0,Y 594.354,Z 747.445,A -85,B 0,C 180,E1 -992.711,E2 -992.711} C_VEL
LIN {X 0,Y 594.335,Z 747.446,A -85,B 0,C 180,E1 -995.428,E2 -995.428} C_VEL
LIN {X 0,Y 594.343,Z 747.456,A -85,B 0,C 180,E1 -998.158,E2 -998.158} C_VEL
LIN {X 0,Y 594.319,Z 747.448,A -85,B 0,C 180,E1 -1001.044,E2 -1001.044} C_VEL
LIN {X 0,Y 594.336,Z 747.447,A -85,B 0,C 180,E1 -1003.68,E2 -1003.68} C_VEL
LIN {X 0,Y 594.382,Z 747.447,A -85,B 0,C 180,E1 -1006.486,E2 -1006.486} C_VEL
LIN {X 0,Y 594.344,Z 747.444,A -85,B 0,C 180,E1 -1009.335,E2 -1009.335} C_VEL
LIN {X 0,Y 594.339,Z 747.445,A -85,B 0,C 180,E1 -1011.504,E2 -1011.504} C_VEL
LIN {X 0,Y 594.378,Z 747.451,A -85,B 0,C 180,E1 -1014.447,E2 -1014.447} C_VEL
LIN {X 0,Y 594.333,Z 747.446,A -85,B 0,C 180,E1 -1017.519,E2 -1017.519} C_VEL
LIN {X 0,Y 594.348,Z 747.445,A -85,B 0,C 180,E1 -1019.778,E2 -1019.778} C_VEL
LIN {X 0,Y 594.356,Z 747.447,A -85,B 0,C 180,E1 -1022.148,E2 -1022.148} C_VEL
LIN {X 0,Y 594.374,Z 747.452,A -85,B 0,C 180,E1 -1024.581,E2 -1024.581} C_VEL
LIN {X 0,Y 594.378,Z 747.44,A -85,B 0,C 180,E1 -1027.609,E2 -1027.609} C_VEL
LIN {X 0,Y 594.355,Z 747.453,A -85,B 0,C 180,E1 -1030.568,E2 -1030.568} C_VEL
LIN {X 0,Y 594.361,Z 747.444,A -85,B 0,C 180,E1 -1033.3,E2 -1033.3} C_VEL
LIN {X 0,Y 594.354,Z 747.445,A -85,B 0,C 180,E1 -1036.162,E2 -1036.162} C_VEL
LIN {X 0,Y 594.371,Z 747.448,A -85,B 0,C 180,E1 -1038.537,E2 -1038.537} C_VEL
LIN {X 0,Y 594.369,Z 747.445,A -85,B 0,C 180,E1 -1041.298,E2 -1041.298} C_VEL
LIN {X 0,Y 594.346,Z 747.444,A -85,B 0,C 180,E1 -1043.756,E2 -1043.756} C_VEL
LIN {X 0,Y 594.3,Z 747.46,A -85,B 0,C 180,E1 -1045.416,E2 -1045.416} C_VEL
LIN {X 0,Y 594.29,Z 750.907,A -85,B 0,C 180,E1 -1048.372,E2 -1048.372} C_VEL
LIN {X 0,Y 594.256,Z 754.206,A -85,B 0,C 180,E1 -1051.065,E2 -1051.065} C_VEL
LIN {X 0,Y 594.287,Z 757.893,A -85,B 0,C 180,E1 -1053.998,E2 -1053.998} C_VEL
LIN {X 0,Y 594.241,Z 760.845,A -85,B 0,C 180,E1 -1056.291,E2 -1056.291} C_VEL
LIN {X 0,Y 594.291,Z 764.688,A -85,B 0,C 180,E1 -1059.221,E2 -1059.221} C_VEL
LIN {X 0,Y 594.217,Z 768.532,A -85,B 0,C 180,E1 -1062.092,E2 -1062.092} C_VEL
LIN {X 0,Y 594.244,Z 771.414,A -85,B 0,C 180,E1 -1064.217,E2 -1064.217} C_VEL
LIN {X 0,Y 594.225,Z 775.258,A -85,B 0,C 180,E1 -1067.015,E2 -1067.015} C_VEL
LIN {X 0,Y 594.272,Z 776.669,A -85,B 0,C 180,E1 -1068.035,E2 -1068.035} C_VEL
LIN {X 0,Y 594.646,Z 782.346,A -85,B 0,C 180,E1 -1068.172,E2 -1068.172} C_VEL
LIN {X 0,Y 594.551,Z 794.142,A -85,B 0,C 180,E1 -1068.495,E2 -1068.495} C_VEL
LIN {X 0,Y 594.537,Z 805.493,A -85,B 0,C 180,E1 -1068.928,E2 -1068.928} C_VEL
LIN {X 0,Y 594.498,Z 817.532,A -85,B 0,C 180,E1 -1069.529,E2 -1069.529} C_VEL
LIN {X 0,Y 594.447,Z 828.33,A -85,B 0,C 180,E1 -1070.216,E2 -1070.216} C_VEL
LIN {X 0,Y 594.404,Z 838.094,A -85,B 0,C 180,E1 -1070.988,E2 -1070.988} C_VEL
LIN {X 0,Y 594.365,Z 846.989,A -85,B 0,C 180,E1 -1071.843,E2 -1071.843} C_VEL
LIN {X 0,Y 594.344,Z 855.669,A -85,B 0,C 180,E1 -1072.868,E2 -1072.868} C_VEL
LIN {X 0,Y 594.29,Z 862.608,A -85,B 0,C 180,E1 -1073.891,E2 -1073.891} C_VEL
LIN {X 0,Y 594.253,Z 868.159,A -85,B 0,C 180,E1 -1074.912,E2 -1074.912} C_VEL
LIN {X 0,Y 594.262,Z 872.519,A -85,B 0,C 180,E1 -1075.932,E2 -1075.932} C_VEL
LIN {X 0,Y 594.268,Z 874.814,A -85,B 0,C 180,E1 -1076.611,E2 -1076.611} C_VEL
LIN {X 0,Y 594.225,Z 876.695,A -85,B 0,C 180,E1 -1077.289,E2 -1077.289} C_VEL
LIN {X 0,Y 594.24,Z 878.13,A -85,B 0,C 180,E1 -1077.967,E2 -1077.967} C_VEL
LIN {X 0,Y 594.24,Z 879.753,A -85,B 0,C 180,E1 -1079.323,E2 -1079.323} C_VEL
LIN {X 0,Y 594.236,Z 879.997,A -85,B 0,C 180,E1 -1080.001,E2 -1080.001} C_VEL
LIN {X 0,Y 594.24,Z 879.816,A -85,B 0,C 180,E1 -1080.678,E2 -1080.678} C_VEL
LIN {X 0,Y 594.239,Z 878.276,A -85,B 0,C 180,E1 -1082.034,E2 -1082.034} C_VEL
LIN {X 0,Y 594.227,Z 876.903,A -85,B 0,C 180,E1 -1082.712,E2 -1082.712} C_VEL
LIN {X 0,Y 594.289,Z 874.026,A -85,B 0,C 180,E1 -1083.73,E2 -1083.73} C_VEL
LIN {X 0,Y 594.241,Z 870.125,A -85,B 0,C 180,E1 -1084.749,E2 -1084.749} C_VEL
LIN {X 0,Y 594.299,Z 865.096,A -85,B 0,C 180,E1 -1085.77,E2 -1085.77} C_VEL
LIN {X 0,Y 594.317,Z 858.782,A -85,B 0,C 180,E1 -1086.792,E2 -1086.792} C_VEL
LIN {X 0,Y 594.347,Z 850.865,A -85,B 0,C 180,E1 -1087.816,E2 -1087.816} C_VEL
LIN {X 0,Y 594.366,Z 842.796,A -85,B 0,C 180,E1 -1088.672,E2 -1088.672} C_VEL
LIN {X 0,Y 594.416,Z 832.948,A -85,B 0,C 180,E1 -1089.528,E2 -1089.528} C_VEL
LIN {X 0,Y 594.469,Z 821.9,A -85,B 0,C 180,E1 -1090.301,E2 -1090.301} C_VEL
LIN {X 0,Y 594.555,Z 809.458,A -85,B 0,C 180,E1 -1090.983,E2 -1090.983} C_VEL
LIN {X 0,Y 594.583,Z 797.925,A -85,B 0,C 180,E1 -1091.467,E2 -1091.467} C_VEL
LIN {X 0,Y 594.632,Z 785.192,A -85,B 0,C 180,E1 -1091.851,E2 -1091.851} C_VEL
LIN {X 0,Y 594.408,Z 778.024,A -85,B 0,C 180,E1 -1092.012,E2 -1092.012} C_VEL
LIN {X 0,Y 594.242,Z 776.642,A -85,B 0,C 180,E1 -1092.075,E2 -1092.075} C_VEL
LIN {X 0,Y 594.238,Z 773.458,A -85,B 0,C 180,E1 -1094.381,E2 -1094.381} C_VEL
LIN {X 0,Y 594.237,Z 769.612,A -85,B 0,C 180,E1 -1097.199,E2 -1097.199} C_VEL
LIN {X 0,Y 594.241,Z 766.729,A -85,B 0,C 180,E1 -1099.339,E2 -1099.339} C_VEL
LIN {X 0,Y 594.226,Z 763.844,A -85,B 0,C 180,E1 -1101.509,E2 -1101.509} C_VEL
LIN {X 0,Y 594.274,Z 759.999,A -85,B 0,C 180,E1 -1104.452,E2 -1104.452} C_VEL
LIN {X 0,Y 594.273,Z 756.105,A -85,B 0,C 180,E1 -1107.505,E2 -1107.505} C_VEL
LIN {X 0,Y 594.27,Z 752.623,A -85,B 0,C 180,E1 -1110.308,E2 -1110.308} C_VEL
LIN {X 0,Y 594.293,Z 749.423,A -85,B 0,C 180,E1 -1112.956,E2 -1112.956} C_VEL
LIN {X 0,Y 594.284,Z 747.797,A -85,B 0,C 180,E1 -1114.124,E2 -1114.124} C_VEL
LIN {X 0,Y 594.28,Z 747.462,A -85,B 0,C 180,E1 -1114.587,E2 -1114.587} C_VEL
LIN {X 0,Y 594.386,Z 747.449,A -85,B 0,C 180,E1 -1117.087,E2 -1117.087} C_VEL
LIN {X 0,Y 594.379,Z 747.442,A -85,B 0,C 180,E1 -1119.774,E2 -1119.774} C_VEL
LIN {X 0,Y 594.352,Z 747.445,A -85,B 0,C 180,E1 -1122.377,E2 -1122.377} C_VEL
LIN {X 0,Y 594.361,Z 747.451,A -85,B 0,C 180,E1 -1125.192,E2 -1125.192} C_VEL
LIN {X 0,Y 594.386,Z 747.441,A -85,B 0,C 180,E1 -1128.152,E2 -1128.152} C_VEL
LIN {X 0,Y 594.384,Z 747.448,A -85,B 0,C 180,E1 -1131.195,E2 -1131.195} C_VEL
LIN {X 0,Y 594.438,Z 747.64,A -85,B 0,C 180,E1 -1133.971,E2 -1133.971} C_VEL
LIN {X 0,Y 594.644,Z 752.263,A -85,B 0,C 180,E1 -1135.437,E2 -1135.437} C_VEL
LIN {X 0,Y 594.613,Z 761.717,A -85,B 0,C 180,E1 -1138.321,E2 -1138.321} C_VEL
LIN {X 0,Y 594.523,Z 770.836,A -85,B 0,C 180,E1 -1141.019,E2 -1141.019} C_VEL
LIN {X 0,Y 594.475,Z 780.035,A -85,B 0,C 180,E1 -1143.673,E2 -1143.673} C_VEL
LIN {X 0,Y 594.453,Z 789.338,A -85,B 0,C 180,E1 -1146.299,E2 -1146.299} C_VEL
LIN {X 0,Y 594.406,Z 799.929,A -85,B 0,C 180,E1 -1149.224,E2 -1149.224} C_VEL
LIN {X 0,Y 594.361,Z 810.52,A -85,B 0,C 180,E1 -1152.095,E2 -1152.095} C_VEL
LIN {X 0,Y 594.301,Z 821.111,A -85,B 0,C 180,E1 -1154.92,E2 -1154.92} C_VEL
LIN {X 0,Y 594.299,Z 831.703,A -85,B 0,C 180,E1 -1157.71,E2 -1157.71} C_VEL
LIN {X 0,Y 594.299,Z 832.53,A -85,B 0,C 180,E1 -1157.926,E2 -1157.926} C_VEL
LIN {X 0,Y 594.677,Z 838.227,A -85,B 0,C 180,E1 -1158.042,E2 -1158.042} C_VEL
LIN {X 0,Y 594.621,Z 851.494,A -85,B 0,C 180,E1 -1158.366,E2 -1158.366} C_VEL
LIN {X 0,Y 594.552,Z 863.417,A -85,B 0,C 180,E1 -1158.792,E2 -1158.792} C_VEL
LIN {X 0,Y 594.512,Z 875.207,A -85,B 0,C 180,E1 -1159.356,E2 -1159.356} C_VEL
LIN {X 0,Y 594.462,Z 886.475,A -85,B 0,C 180,E1 -1160.043,E2 -1160.043} C_VEL
LIN {X 0,Y 594.406,Z 896.646,A -85,B 0,C 180,E1 -1160.815,E2 -1160.815} C_VEL
LIN {X 0,Y 594.373,Z 905.787,A -85,B 0,C 180,E1 -1161.672,E2 -1161.672} C_VEL
LIN {X 0,Y 594.317,Z 914.691,A -85,B 0,C 180,E1 -1162.697,E2 -1162.697} C_VEL
LIN {X 0,Y 594.281,Z 921.171,A -85,B 0,C 180,E1 -1163.615,E2 -1163.615} C_VEL
LIN {X 0,Y 594.289,Z 926.68,A -85,B 0,C 180,E1 -1164.571,E2 -1164.571} C_VEL
LIN {X 0,Y 594.27,Z 931.371,A -85,B 0,C 180,E1 -1165.591,E2 -1165.591} C_VEL
LIN {X 0,Y 594.268,Z 934.956,A -85,B 0,C 180,E1 -1166.61,E2 -1166.61} C_VEL
LIN {X 0,Y 594.226,Z 936.809,A -85,B 0,C 180,E1 -1167.288,E2 -1167.288} C_VEL
LIN {X 0,Y 594.239,Z 938.202,A -85,B 0,C 180,E1 -1167.967,E2 -1167.967} C_VEL
LIN {X 0,Y 594.239,Z 939.784,A -85,B 0,C 180,E1 -1169.322,E2 -1169.322} C_VEL
LIN {X 0,Y 594.236,Z 940,A -85,B 0,C 180,E1 -1170,E2 -1170} C_VEL
LIN {X 0,Y 594.247,Z 939.184,A -85,B 0,C 180,E1 -1171.355,E2 -1171.355} C_VEL
LIN {X 0,Y 594.239,Z 938.202,A -85,B 0,C 180,E1 -1172.033,E2 -1172.033} C_VEL
LIN {X 0,Y 594.226,Z 936.809,A -85,B 0,C 180,E1 -1172.712,E2 -1172.712} C_VEL
LIN {X 0,Y 594.289,Z 933.896,A -85,B 0,C 180,E1 -1173.729,E2 -1173.729} C_VEL
LIN {X 0,Y 594.241,Z 929.95,A -85,B 0,C 180,E1 -1174.749,E2 -1174.749} C_VEL
LIN {X 0,Y 594.304,Z 923.877,A -85,B 0,C 180,E1 -1175.939,E2 -1175.939} C_VEL
LIN {X 0,Y 594.308,Z 917.235,A -85,B 0,C 180,E1 -1176.962,E2 -1176.962} C_VEL
LIN {X 0,Y 594.359,Z 908.989,A -85,B 0,C 180,E1 -1177.986,E2 -1177.986} C_VEL
LIN {X 0,Y 594.382,Z 900.536,A -85,B 0,C 180,E1 -1178.842,E2 -1178.842} C_VEL
LIN {X 0,Y 594.429,Z 890.092,A -85,B 0,C 180,E1 -1179.699,E2 -1179.699} C_VEL
LIN {X 0,Y 594.487,Z 879.757,A -85,B 0,C 180,E1 -1180.386,E2 -1180.386} C_VEL
LIN {X 0,Y 594.521,Z 867.597,A -85,B 0,C 180,E1 -1181.026,E2 -1181.026} C_VEL
LIN {X 0,Y 594.589,Z 855.461,A -85,B 0,C 180,E1 -1181.506,E2 -1181.506} C_VEL
LIN {X 0,Y 594.652,Z 842.435,A -85,B 0,C 180,E1 -1181.872,E2 -1181.872} C_VEL
LIN {X 0,Y 594.467,Z 833.858,A -85,B 0,C 180,E1 -1182.038,E2 -1182.038} C_VEL
LIN {X 0,Y 594.299,Z 832.53,A -85,B 0,C 180,E1 -1182.074,E2 -1182.074} C_VEL
LIN {X 0,Y 594.312,Z 822.435,A -85,B 0,C 180,E1 -1184.729,E2 -1184.729} C_VEL
LIN {X 0,Y 594.335,Z 811.844,A -85,B 0,C 180,E1 -1187.55,E2 -1187.55} C_VEL
LIN {X 0,Y 594.383,Z 801.253,A -85,B 0,C 180,E1 -1190.415,E2 -1190.415} C_VEL
LIN {X 0,Y 594.442,Z 790.661,A -85,B 0,C 180,E1 -1193.333,E2 -1193.333} C_VEL
LIN {X 0,Y 594.489,Z 781.031,A -85,B 0,C 180,E1 -1196.042,E2 -1196.042} C_VEL
LIN {X 0,Y 594.508,Z 772.143,A -85,B 0,C 180,E1 -1198.601,E2 -1198.601} C_VEL
LIN {X 0,Y 594.592,Z 762.859,A -85,B 0,C 180,E1 -1201.337,E2 -1201.337} C_VEL
LIN {X 0,Y 594.657,Z 753.489,A -85,B 0,C 180,E1 -1204.177,E2 -1204.177} C_VEL
LIN {X 0,Y 594.553,Z 748.389,A -85,B 0,C 180,E1 -1205.812,E2 -1205.812} C_VEL
LIN {X 0,Y 594.39,Z 747.448,A -85,B 0,C 180,E1 -1206.19,E2 -1206.19} C_VEL
LIN {X 0,Y 594.384,Z 747.448,A -85,B 0,C 180,E1 -1208.805,E2 -1208.805} C_VEL
LIN {X 0,Y 594.386,Z 747.441,A -85,B 0,C 180,E1 -1211.848,E2 -1211.848} C_VEL
LIN {X 0,Y 594.361,Z 747.451,A -85,B 0,C 180,E1 -1214.808,E2 -1214.808} C_VEL
LIN {X 0,Y 594.351,Z 747.446,A -85,B 0,C 180,E1 -1217.623,E2 -1217.623} C_VEL
LIN {X 0,Y 594.378,Z 747.443,A -85,B 0,C 180,E1 -1220.319,E2 -1220.319} C_VEL
LIN {X 0,Y 594.385,Z 747.451,A -85,B 0,C 180,E1 -1222.913,E2 -1222.913} C_VEL
LIN {X 0,Y 594.305,Z 747.62,A -85,B 0,C 180,E1 -1225.415,E2 -1225.415} C_VEL
LIN {X 0,Y 594.268,Z 750.276,A -85,B 0,C 180,E1 -1227.846,E2 -1227.846} C_VEL
LIN {X 0,Y 594.244,Z 753.158,A -85,B 0,C 180,E1 -1230.216,E2 -1230.216} C_VEL
LIN {X 0,Y 594.267,Z 756.04,A -85,B 0,C 180,E1 -1232.533,E2 -1232.533} C_VEL
LIN {X 0,Y 594.275,Z 759.938,A -85,B 0,C 180,E1 -1235.591,E2 -1235.591} C_VEL
LIN {X 0,Y 594.219,Z 763.726,A -85,B 0,C 180,E1 -1238.491,E2 -1238.491} C_VEL
LIN {X 0,Y 594.245,Z 767.211,A -85,B 0,C 180,E1 -1241.111,E2 -1241.111} C_VEL
LIN {X 0,Y 594.248,Z 770.451,A -85,B 0,C 180,E1 -1243.51,E2 -1243.51} C_VEL
LIN {X 0,Y 594.237,Z 774.295,A -85,B 0,C 180,E1 -1246.317,E2 -1246.317} C_VEL
LIN {X 0,Y 594.255,Z 776.667,A -85,B 0,C 180,E1 -1248.033,E2 -1248.033} C_VEL
LIN {X 0,Y 594.643,Z 781.421,A -85,B 0,C 180,E1 -1248.149,E2 -1248.149} C_VEL
LIN {X 0,Y 594.603,Z 794.018,A -85,B 0,C 180,E1 -1248.491,E2 -1248.491} C_VEL
LIN {X 0,Y 594.563,Z 805.822,A -85,B 0,C 180,E1 -1248.942,E2 -1248.942} C_VEL
LIN {X 0,Y 594.51,Z 817.512,A -85,B 0,C 180,E1 -1249.527,E2 -1249.527} C_VEL
LIN {X 0,Y 594.437,Z 828.309,A -85,B 0,C 180,E1 -1250.214,E2 -1250.214} C_VEL
LIN {X 0,Y 594.405,Z 838.083,A -85,B 0,C 180,E1 -1250.986,E2 -1250.986} C_VEL
LIN {X 0,Y 594.366,Z 846.98,A -85,B 0,C 180,E1 -1251.842,E2 -1251.842} C_VEL
LIN {X 0,Y 594.308,Z 855.666,A -85,B 0,C 180,E1 -1252.867,E2 -1252.867} C_VEL
LIN {X 0,Y 594.29,Z 862.596,A -85,B 0,C 180,E1 -1253.89,E2 -1253.89} C_VEL
LIN {X 0,Y 594.254,Z 868.148,A -85,B 0,C 180,E1 -1254.911,E2 -1254.911} C_VEL
LIN {X 0,Y 594.262,Z 872.511,A -85,B 0,C 180,E1 -1255.93,E2 -1255.93} C_VEL
LIN {X 0,Y 594.267,Z 874.814,A -85,B 0,C 180,E1 -1256.609,E2 -1256.609} C_VEL
LIN {X 0,Y 594.227,Z 876.692,A -85,B 0,C 180,E1 -1257.288,E2 -1257.288} C_VEL
LIN {X 0,Y 594.24,Z 878.127,A -85,B 0,C 180,E1 -1257.966,E2 -1257.966} C_VEL
LIN {X 0,Y 594.241,Z 879.753,A -85,B 0,C 180,E1 -1259.322,E2 -1259.322} C_VEL
LIN {X 0,Y 594.236,Z 879.995,A -85,B 0,C 180,E1 -1259.999,E2 -1259.999} C_VEL
LIN {X 0,Y 594.239,Z 879.815,A -85,B 0,C 180,E1 -1260.677,E2 -1260.677} C_VEL
LIN {X 0,Y 594.24,Z 878.276,A -85,B 0,C 180,E1 -1262.033,E2 -1262.033} C_VEL
LIN {X 0,Y 594.226,Z 876.917,A -85,B 0,C 180,E1 -1262.711,E2 -1262.711} C_VEL
LIN {X 0,Y 594.29,Z 874.04,A -85,B 0,C 180,E1 -1263.729,E2 -1263.729} C_VEL
LIN {X 0,Y 594.241,Z 870.141,A -85,B 0,C 180,E1 -1264.748,E2 -1264.748} C_VEL
LIN {X 0,Y 594.299,Z 865.111,A -85,B 0,C 180,E1 -1265.768,E2 -1265.768} C_VEL
LIN {X 0,Y 594.315,Z 858.793,A -85,B 0,C 180,E1 -1266.791,E2 -1266.791} C_VEL
LIN {X 0,Y 594.346,Z 850.876,A -85,B 0,C 180,E1 -1267.815,E2 -1267.815} C_VEL
LIN {X 0,Y 594.381,Z 841.032,A -85,B 0,C 180,E1 -1268.841,E2 -1268.841} C_VEL
LIN {X 0,Y 594.434,Z 830.711,A -85,B 0,C 180,E1 -1269.699,E2 -1269.699} C_VEL
LIN {X 0,Y 594.498,Z 819.093,A -85,B 0,C 180,E1 -1270.471,E2 -1270.471} C_VEL
LIN {X 0,Y 594.535,Z 807.582,A -85,B 0,C 180,E1 -1271.072,E2 -1271.072} C_VEL
LIN {X 0,Y 594.542,Z 795.444,A -85,B 0,C 180,E1 -1271.552,E2 -1271.552} C_VEL
LIN {X 0,Y 594.638,Z 786.742,A -85,B 0,C 180,E1 -1271.814,E2 -1271.814} C_VEL
LIN {X 0,Y 594.247,Z 783.403,A -85,B 0,C 180,E1 -1271.969,E2 -1271.969} C_VEL
LIN {X 0,Y 593.342,Z 780.699,A -85,B 0,C 180,E1 -1272.209,E2 -1272.209} C_VEL
LIN {X 0,Y 591.506,Z 777.723,A -85,B 0,C 180,E1 -1272.663,E2 -1272.663} C_VEL
LIN {X 0,Y 588.884,Z 775.339,A -85,B 0,C 180,E1 -1273.396,E2 -1273.396} C_VEL
LIN {X 0,Y 587.234,Z 773.953,A -85,B 0,C 180,E1 -1274.196,E2 -1274.196} C_VEL
LIN {X 0,Y 587.136,Z 773.672,A -85,B 0,C 180,E1 -1274.401,E2 -1274.401} C_VEL
LIN {X 0,Y 587.144,Z 770.504,A -85,B 0,C 180,E1 -1276.747,E2 -1276.747} C_VEL
LIN {X 0,Y 587.115,Z 766.73,A -85,B 0,C 180,E1 -1279.582,E2 -1279.582} C_VEL
LIN {X 0,Y 587.141,Z 763.846,A -85,B 0,C 180,E1 -1281.78,E2 -1281.78} C_VEL
LIN {X 0,Y 587.176,Z 760,A -85,B 0,C 180,E1 -1284.765,E2 -1284.765} C_VEL
LIN {X 0,Y 587.163,Z 757.116,A -85,B 0,C 180,E1 -1287.053,E2 -1287.053} C_VEL
LIN {X 0,Y 587.162,Z 754.231,A -85,B 0,C 180,E1 -1289.389,E2 -1289.389} C_VEL
LIN {X 0,Y 587.217,Z 751.299,A -85,B 0,C 180,E1 -1291.815,E2 -1291.815} C_VEL
LIN {X 0,Y 587.224,Z 748.419,A -85,B 0,C 180,E1 -1294.33,E2 -1294.33} C_VEL
LIN {X 0,Y 587.346,Z 748.32,A -85,B 0,C 180,E1 -1296.746,E2 -1296.746} C_VEL
LIN {X 0,Y 587.325,Z 748.328,A -85,B 0,C 180,E1 -1299.36,E2 -1299.36} C_VEL
LIN {X 0,Y 587.331,Z 748.319,A -85,B 0,C 180,E1 -1302.107,E2 -1302.107} C_VEL
LIN {X 0,Y 587.312,Z 748.327,A -85,B 0,C 180,E1 -1305.088,E2 -1305.088} C_VEL
LIN {X 0,Y 587.313,Z 748.323,A -85,B 0,C 180,E1 -1307.924,E2 -1307.924} C_VEL
LIN {X 0,Y 587.324,Z 748.32,A -85,B 0,C 180,E1 -1310.639,E2 -1310.639} C_VEL
LIN {X 0,Y 587.342,Z 748.324,A -85,B 0,C 180,E1 -1313.292,E2 -1313.292} C_VEL
LIN {X 0,Y 587.325,Z 748.325,A -85,B 0,C 180,E1 -1315.777,E2 -1315.777} C_VEL
LIN {X 0,Y 587.331,Z 748.319,A -85,B 0,C 180,E1 -1318.23,E2 -1318.23} C_VEL
LIN {X 0,Y 587.34,Z 748.318,A -85,B 0,C 180,E1 -1320.866,E2 -1320.866} C_VEL
LIN {X 0,Y 587.322,Z 748.327,A -85,B 0,C 180,E1 -1323.824,E2 -1323.824} C_VEL
LIN {X 0,Y 587.304,Z 748.327,A -85,B 0,C 180,E1 -1325.992,E2 -1325.992} C_VEL
LIN {X 0,Y 587.303,Z 748.324,A -85,B 0,C 180,E1 -1328.225,E2 -1328.225} C_VEL
LIN {X 0,Y 587.337,Z 748.319,A -85,B 0,C 180,E1 -1331.151,E2 -1331.151} C_VEL
LIN {X 0,Y 587.299,Z 748.329,A -85,B 0,C 180,E1 -1334.024,E2 -1334.024} C_VEL
LIN {X 0,Y 587.335,Z 748.323,A -85,B 0,C 180,E1 -1336.154,E2 -1336.154} C_VEL
LIN {X 0,Y 587.327,Z 748.319,A -85,B 0,C 180,E1 -1338.962,E2 -1338.962} C_VEL
LIN {X 0,Y 587.324,Z 748.327,A -85,B 0,C 180,E1 -1341.744,E2 -1341.744} C_VEL
LIN {X 0,Y 587.313,Z 748.322,A -85,B 0,C 180,E1 -1344.507,E2 -1344.507} C_VEL
LIN {X 0,Y 587.324,Z 748.32,A -85,B 0,C 180,E1 -1347.257,E2 -1347.257} C_VEL
LIN {X 0,Y 587.37,Z 748.323,A -85,B 0,C 180,E1 -1350,E2 -1350} C_VEL
LIN {X 0,Y 587.322,Z 748.32,A -85,B 0,C 180,E1 -1352.744,E2 -1352.744} C_VEL
LIN {X 0,Y 587.305,Z 748.323,A -85,B 0,C 180,E1 -1355.493,E2 -1355.493} C_VEL
LIN {X 0,Y 587.307,Z 748.33,A -85,B 0,C 180,E1 -1358.256,E2 -1358.256} C_VEL
LIN {X 0,Y 587.285,Z 748.324,A -85,B 0,C 180,E1 -1361.107,E2 -1361.107} C_VEL
LIN {X 0,Y 587.323,Z 748.323,A -85,B 0,C 180,E1 -1363.847,E2 -1363.847} C_VEL
LIN {X 0,Y 587.303,Z 748.324,A -85,B 0,C 180,E1 -1366.803,E2 -1366.803} C_VEL
LIN {X 0,Y 587.292,Z 748.324,A -85,B 0,C 180,E1 -1369.577,E2 -1369.577} C_VEL
LIN {X 0,Y 587.299,Z 748.324,A -85,B 0,C 180,E1 -1371.775,E2 -1371.775} C_VEL
LIN {X 0,Y 587.305,Z 748.326,A -85,B 0,C 180,E1 -1374.761,E2 -1374.761} C_VEL
LIN {X 0,Y 587.292,Z 748.324,A -85,B 0,C 180,E1 -1377.684,E2 -1377.684} C_VEL
LIN {X 0,Y 587.307,Z 748.326,A -85,B 0,C 180,E1 -1380.172,E2 -1380.172} C_VEL
LIN {X 0,Y 587.329,Z 748.329,A -85,B 0,C 180,E1 -1382.58,E2 -1382.58} C_VEL
LIN {X 0,Y 587.318,Z 748.323,A -85,B 0,C 180,E1 -1385.056,E2 -1385.056} C_VEL
LIN {X 0,Y 587.325,Z 748.319,A -85,B 0,C 180,E1 -1387.838,E2 -1387.838} C_VEL
LIN {X 0,Y 587.301,Z 748.326,A -85,B 0,C 180,E1 -1390.256,E2 -1390.256} C_VEL
LIN {X 0,Y 587.309,Z 748.325,A -85,B 0,C 180,E1 -1393.119,E2 -1393.119} C_VEL
LIN {X 0,Y 587.307,Z 748.322,A -85,B 0,C 180,E1 -1396.049,E2 -1396.049} C_VEL
LIN {X 0,Y 587.331,Z 748.327,A -85,B 0,C 180,E1 -1398.926,E2 -1398.926} C_VEL
LIN {X 0,Y 587.317,Z 748.321,A -85,B 0,C 180,E1 -1401.521,E2 -1401.521} C_VEL
LIN {X 0,Y 587.286,Z 748.325,A -85,B 0,C 180,E1 -1404.101,E2 -1404.101} C_VEL
LIN {X 0,Y 587.217,Z 748.342,A -85,B 0,C 180,E1 -1405.772,E2 -1405.772} C_VEL
LIN {X 0,Y 587.201,Z 751.24,A -85,B 0,C 180,E1 -1408.224,E2 -1408.224} C_VEL
LIN {X 0,Y 587.167,Z 754.473,A -85,B 0,C 180,E1 -1410.899,E2 -1410.899} C_VEL
LIN {X 0,Y 587.211,Z 758.131,A -85,B 0,C 180,E1 -1413.849,E2 -1413.849} C_VEL
LIN {X 0,Y 587.152,Z 761.807,A -85,B 0,C 180,E1 -1416.735,E2 -1416.735} C_VEL
LIN {X 0,Y 587.167,Z 765.65,A -85,B 0,C 180,E1 -1419.69,E2 -1419.69} C_VEL
LIN {X 0,Y 587.131,Z 769.493,A -85,B 0,C 180,E1 -1422.588,E2 -1422.588} C_VEL
LIN {X 0,Y 587.132,Z 772.376,A -85,B 0,C 180,E1 -1424.732,E2 -1424.732} C_VEL
LIN {X 0,Y 587.13,Z 775.258,A -85,B 0,C 180,E1 -1426.855,E2 -1426.855} C_VEL
LIN {X 0,Y 587.159,Z 776.67,A -85,B 0,C 180,E1 -1427.888,E2 -1427.888} C_VEL
LIN {X 0,Y 587.726,Z 781.437,A -85,B 0,C 180,E1 -1428.009,E2 -1428.009} C_VEL
LIN {X 0,Y 587.612,Z 794.285,A -85,B 0,C 180,E1 -1428.362,E2 -1428.362} C_VEL
LIN {X 0,Y 587.561,Z 806.429,A -85,B 0,C 180,E1 -1428.835,E2 -1428.835} C_VEL
LIN {X 0,Y 587.522,Z 817.541,A -85,B 0,C 180,E1 -1429.403,E2 -1429.403} C_VEL
LIN {X 0,Y 587.445,Z 828.337,A -85,B 0,C 180,E1 -1430.098,E2 -1430.098} C_VEL
LIN {X 0,Y 587.357,Z 838.099,A -85,B 0,C 180,E1 -1430.878,E2 -1430.878} C_VEL
LIN {X 0,Y 587.302,Z 846.992,A -85,B 0,C 180,E1 -1431.745,E2 -1431.745} C_VEL
LIN {X 0,Y 587.259,Z 854.335,A -85,B 0,C 180,E1 -1432.609,E2 -1432.609} C_VEL
LIN {X 0,Y 587.198,Z 861.424,A -85,B 0,C 180,E1 -1433.625,E2 -1433.625} C_VEL
LIN {X 0,Y 587.211,Z 866.432,A -85,B 0,C 180,E1 -1434.506,E2 -1434.506} C_VEL
LIN {X 0,Y 587.188,Z 871.178,A -85,B 0,C 180,E1 -1435.539,E2 -1435.539} C_VEL
LIN {X 0,Y 587.194,Z 874.815,A -85,B 0,C 180,E1 -1436.57,E2 -1436.57} C_VEL
LIN {X 0,Y 587.131,Z 876.693,A -85,B 0,C 180,E1 -1437.256,E2 -1437.256} C_VEL
LIN {X 0,Y 587.139,Z 878.132,A -85,B 0,C 180,E1 -1437.943,E2 -1437.943} C_VEL
LIN {X 0,Y 587.14,Z 879.753,A -85,B 0,C 180,E1 -1439.315,E2 -1439.315} C_VEL
LIN {X 0,Y 587.137,Z 879.997,A -85,B 0,C 180,E1 -1440.001,E2 -1440.001} C_VEL
LIN {X 0,Y 587.14,Z 879.815,A -85,B 0,C 180,E1 -1440.687,E2 -1440.687} C_VEL
LIN {X 0,Y 587.138,Z 878.276,A -85,B 0,C 180,E1 -1442.059,E2 -1442.059} C_VEL
LIN {X 0,Y 587.133,Z 876.896,A -85,B 0,C 180,E1 -1442.745,E2 -1442.745} C_VEL
LIN {X 0,Y 587.213,Z 874.019,A -85,B 0,C 180,E1 -1443.775,E2 -1443.775} C_VEL
LIN {X 0,Y 587.146,Z 870.119,A -85,B 0,C 180,E1 -1444.807,E2 -1444.807} C_VEL
LIN {X 0,Y 587.229,Z 865.091,A -85,B 0,C 180,E1 -1445.839,E2 -1445.839} C_VEL
LIN {X 0,Y 587.231,Z 858.777,A -85,B 0,C 180,E1 -1446.874,E2 -1446.874} C_VEL
LIN {X 0,Y 587.288,Z 850.861,A -85,B 0,C 180,E1 -1447.911,E2 -1447.911} C_VEL
LIN {X 0,Y 587.325,Z 842.791,A -85,B 0,C 180,E1 -1448.776,E2 -1448.776} C_VEL
LIN {X 0,Y 587.386,Z 832.932,A -85,B 0,C 180,E1 -1449.644,E2 -1449.644} C_VEL
LIN {X 0,Y 587.481,Z 821.893,A -85,B 0,C 180,E1 -1450.425,E2 -1450.425} C_VEL
LIN {X 0,Y 587.571,Z 808.898,A -85,B 0,C 180,E1 -1451.142,E2 -1451.142} C_VEL
LIN {X 0,Y 587.618,Z 796.85,A -85,B 0,C 180,E1 -1451.64,E2 -1451.64} C_VEL
LIN {X 0,Y 587.687,Z 784.249,A -85,B 0,C 180,E1 -1452.015,E2 -1452.015} C_VEL
LIN {X 0,Y 587.477,Z 778.861,A -85,B 0,C 180,E1 -1452.14,E2 -1452.14} C_VEL
LIN {X 0,Y 587.143,Z 776.671,A -85,B 0,C 180,E1 -1452.202,E2 -1452.202} C_VEL
LIN {X 0,Y 587.132,Z 773.457,A -85,B 0,C 180,E1 -1454.559,E2 -1454.559} C_VEL
LIN {X 0,Y 587.148,Z 770.503,A -85,B 0,C 180,E1 -1456.748,E2 -1456.748} C_VEL
LIN {X 0,Y 587.134,Z 766.728,A -85,B 0,C 180,E1 -1459.583,E2 -1459.583} C_VEL
LIN {X 0,Y 587.143,Z 763.844,A -85,B 0,C 180,E1 -1461.782,E2 -1461.782} C_VEL
LIN {X 0,Y 587.174,Z 759.998,A -85,B 0,C 180,E1 -1464.767,E2 -1464.767} C_VEL
LIN {X 0,Y 587.188,Z 756.152,A -85,B 0,C 180,E1 -1467.827,E2 -1467.827} C_VEL
LIN {X 0,Y 587.198,Z 752.306,A -85,B 0,C 180,E1 -1470.975,E2 -1470.975} C_VEL
LIN {X 0,Y 587.183,Z 749.118,A -85,B 0,C 180,E1 -1473.407,E2 -1473.407} C_VEL
LIN {X 0,Y 587.234,Z 748.341,A -85,B 0,C 180,E1 -1474.331,E2 -1474.331} C_VEL
LIN {X 0,Y 587.324,Z 748.324,A -85,B 0,C 180,E1 -1476.749,E2 -1476.749} C_VEL
LIN {X 0,Y 587.347,Z 748.323,A -85,B 0,C 180,E1 -1479.36,E2 -1479.36} C_VEL
LIN {X 0,Y 587.314,Z 748.321,A -85,B 0,C 180,E1 -1482.105,E2 -1482.105} C_VEL
LIN {X 0,Y 587.311,Z 748.331,A -85,B 0,C 180,E1 -1485.088,E2 -1485.088} C_VEL
LIN {X 0,Y 587.329,Z 748.319,A -85,B 0,C 180,E1 -1487.925,E2 -1487.925} C_VEL
LIN {X 0,Y 587.337,Z 748.325,A -85,B 0,C 180,E1 -1490.64,E2 -1490.64} C_VEL
LIN {X 0,Y 587.354,Z 748.323,A -85,B 0,C 180,E1 -1493.292,E2 -1493.292} C_VEL
LIN {X 0,Y 587.36,Z 748.476,A -85,B 0,C 180,E1 -1493.733,E2 -1493.733} C_VEL
LIN {X 0,Y 587.705,Z 752.251,A -85,B 0,C 180,E1 -1494.97,E2 -1494.97} C_VEL
LIN {X 0,Y 587.666,Z 761.448,A -85,B 0,C 180,E1 -1497.82,E2 -1497.82} C_VEL
LIN {X 0,Y 587.569,Z 770.803,A -85,B 0,C 180,E1 -1500.633,E2 -1500.633} C_VEL
LIN {X 0,Y 587.502,Z 780.07,A -85,B 0,C 180,E1 -1503.346,E2 -1503.346} C_VEL
LIN {X 0,Y 587.436,Z 790.661,A -85,B 0,C 180,E1 -1506.372,E2 -1506.372} C_VEL
LIN {X 0,Y 587.377,Z 801.253,A -85,B 0,C 180,E1 -1509.331,E2 -1509.331} C_VEL
LIN {X 0,Y 587.303,Z 811.844,A -85,B 0,C 180,E1 -1512.233,E2 -1512.233} C_VEL
LIN {X 0,Y 587.257,Z 822.435,A -85,B 0,C 180,E1 -1515.09,E2 -1515.09} C_VEL
LIN {X 0,Y 587.216,Z 832.571,A -85,B 0,C 180,E1 -1517.789,E2 -1517.789} C_VEL
LIN {X 0,Y 587.736,Z 838.227,A -85,B 0,C 180,E1 -1517.899,E2 -1517.899} C_VEL
LIN {X 0,Y 587.686,Z 851.494,A -85,B 0,C 180,E1 -1518.226,E2 -1518.226} C_VEL
LIN {X 0,Y 587.576,Z 863.387,A -85,B 0,C 180,E1 -1518.655,E2 -1518.655} C_VEL
LIN {X 0,Y 587.527,Z 875.208,A -85,B 0,C 180,E1 -1519.228,E2 -1519.228} C_VEL
LIN {X 0,Y 587.451,Z 886.476,A -85,B 0,C 180,E1 -1519.923,E2 -1519.923} C_VEL
LIN {X 0,Y 587.384,Z 896.646,A -85,B 0,C 180,E1 -1520.704,E2 -1520.704} C_VEL
LIN {X 0,Y 587.34,Z 905.787,A -85,B 0,C 180,E1 -1521.571,E2 -1521.571} C_VEL
LIN {X 0,Y 587.259,Z 914.69,A -85,B 0,C 180,E1 -1522.608,E2 -1522.608} C_VEL
LIN {X 0,Y 587.195,Z 921.748,A -85,B 0,C 180,E1 -1523.627,E2 -1523.627} C_VEL
LIN {X 0,Y 587.211,Z 926.68,A -85,B 0,C 180,E1 -1524.506,E2 -1524.506} C_VEL
LIN {X 0,Y 587.189,Z 931.371,A -85,B 0,C 180,E1 -1525.538,E2 -1525.538} C_VEL
LIN {X 0,Y 587.194,Z 934.956,A -85,B 0,C 180,E1 -1526.569,E2 -1526.569} C_VEL
LIN {X 0,Y 587.132,Z 936.809,A -85,B 0,C 180,E1 -1527.256,E2 -1527.256} C_VEL
LIN {X 0,Y 587.138,Z 938.201,A -85,B 0,C 180,E1 -1527.942,E2 -1527.942} C_VEL
LIN {X 0,Y 587.14,Z 939.784,A -85,B 0,C 180,E1 -1529.314,E2 -1529.314} C_VEL
LIN {X 0,Y 587.137,Z 940,A -85,B 0,C 180,E1 -1530,E2 -1530} C_VEL
LIN {X 0,Y 587.147,Z 939.185,A -85,B 0,C 180,E1 -1531.372,E2 -1531.372} C_VEL
LIN {X 0,Y 587.138,Z 938.202,A -85,B 0,C 180,E1 -1532.058,E2 -1532.058} C_VEL
LIN {X 0,Y 587.132,Z 936.809,A -85,B 0,C 180,E1 -1532.744,E2 -1532.744} C_VEL
LIN {X 0,Y 587.213,Z 933.896,A -85,B 0,C 180,E1 -1533.774,E2 -1533.774} C_VEL
LIN {X 0,Y 587.147,Z 929.95,A -85,B 0,C 180,E1 -1534.806,E2 -1534.806} C_VEL
LIN {X 0,Y 587.217,Z 923.877,A -85,B 0,C 180,E1 -1536.011,E2 -1536.011} C_VEL
LIN {X 0,Y 587.245,Z 917.236,A -85,B 0,C 180,E1 -1537.046,E2 -1537.046} C_VEL
LIN {X 0,Y 587.3,Z 908.989,A -85,B 0,C 180,E1 -1538.083,E2 -1538.083} C_VEL
LIN {X 0,Y 587.343,Z 900.537,A -85,B 0,C 180,E1 -1538.949,E2 -1538.949} C_VEL
LIN {X 0,Y 587.415,Z 890.093,A -85,B 0,C 180,E1 -1539.816,E2 -1539.816} C_VEL
LIN {X 0,Y 587.504,Z 879.758,A -85,B 0,C 180,E1 -1540.511,E2 -1540.511} C_VEL
LIN {X 0,Y 587.537,Z 868.083,A -85,B 0,C 180,E1 -1541.137,E2 -1541.137} C_VEL
LIN {X 0,Y 587.629,Z 855.65,A -85,B 0,C 180,E1 -1541.637,E2 -1541.637} C_VEL
LIN {X 0,Y 587.721,Z 842.434,A -85,B 0,C 180,E1 -1542.014,E2 -1542.014} C_VEL
LIN {X 0,Y 587.447,Z 834.233,A -85,B 0,C 180,E1 -1542.178,E2 -1542.178} C_VEL
LIN {X 0,Y 587.216,Z 832.53,A -85,B 0,C 180,E1 -1542.221,E2 -1542.221} C_VEL
LIN {X 0,Y 587.257,Z 822.435,A -85,B 0,C 180,E1 -1544.91,E2 -1544.91} C_VEL
LIN {X 0,Y 587.303,Z 811.844,A -85,B 0,C 180,E1 -1547.767,E2 -1547.767} C_VEL
LIN {X 0,Y 587.377,Z 801.253,A -85,B 0,C 180,E1 -1550.669,E2 -1550.669} C_VEL
LIN {X 0,Y 587.436,Z 790.661,A -85,B 0,C 180,E1 -1553.628,E2 -1553.628} C_VEL
LIN {X 0,Y 587.502,Z 780.07,A -85,B 0,C 180,E1 -1556.654,E2 -1556.654} C_VEL
LIN {X 0,Y 587.569,Z 770.803,A -85,B 0,C 180,E1 -1559.367,E2 -1559.367} C_VEL
LIN {X 0,Y 587.666,Z 761.448,A -85,B 0,C 180,E1 -1562.18,E2 -1562.18} C_VEL
LIN {X 0,Y 587.692,Z 754.215,A -85,B 0,C 180,E1 -1564.396,E2 -1564.396} C_VEL
LIN {X 0,Y 587.588,Z 749.735,A -85,B 0,C 180,E1 -1565.879,E2 -1565.879} C_VEL
LIN {X 0,Y 587.345,Z 748.326,A -85,B 0,C 180,E1 -1566.418,E2 -1566.418} C_VEL
LIN {X 0,Y 587.337,Z 748.326,A -85,B 0,C 180,E1 -1569.36,E2 -1569.36} C_VEL
LIN {X 0,Y 587.34,Z 748.319,A -85,B 0,C 180,E1 -1572.108,E2 -1572.108} C_VEL
LIN {X 0,Y 587.306,Z 748.332,A -85,B 0,C 180,E1 -1575.087,E2 -1575.087} C_VEL
LIN {X 0,Y 587.315,Z 748.322,A -85,B 0,C 180,E1 -1577.924,E2 -1577.924} C_VEL
LIN {X 0,Y 587.335,Z 748.325,A -85,B 0,C 180,E1 -1580.639,E2 -1580.639} C_VEL
LIN {X 0,Y 587.323,Z 748.325,A -85,B 0,C 180,E1 -1583.296,E2 -1583.296} C_VEL
LIN {X 0,Y 587.28,Z 748.336,A -85,B 0,C 180,E1 -1584.941,E2 -1584.941} C_VEL
LIN {X 0,Y 587.262,Z 748.711,A -85,B 0,C 180,E1 -1585.773,E2 -1585.773} C_VEL
LIN {X 0,Y 587.193,Z 751.238,A -85,B 0,C 180,E1 -1588.222,E2 -1588.222} C_VEL
LIN {X 0,Y 587.169,Z 754.472,A -85,B 0,C 180,E1 -1590.899,E2 -1590.899} C_VEL
LIN {X 0,Y 587.163,Z 757.001,A -85,B 0,C 180,E1 -1592.945,E2 -1592.945} C_VEL
LIN {X 0,Y 587.173,Z 760.844,A -85,B 0,C 180,E1 -1595.986,E2 -1595.986} C_VEL
LIN {X 0,Y 587.181,Z 764.746,A -85,B 0,C 180,E1 -1599.002,E2 -1599.002} C_VEL
LIN {X 0,Y 587.126,Z 768.531,A -85,B 0,C 180,E1 -1601.866,E2 -1601.866} C_VEL
LIN {X 0,Y 587.153,Z 771.413,A -85,B 0,C 180,E1 -1604.019,E2 -1604.019} C_VEL
LIN {X 0,Y 587.136,Z 775.257,A -85,B 0,C 180,E1 -1606.854,E2 -1606.854} C_VEL
LIN {X 0,Y 587.133,Z 776.668,A -85,B 0,C 180,E1 -1607.886,E2 -1607.886} C_VEL
LIN {X 0,Y 587.696,Z 782.36,A -85,B 0,C 180,E1 -1608.029,E2 -1608.029} C_VEL
LIN {X 0,Y 587.629,Z 795.574,A -85,B 0,C 180,E1 -1608.405,E2 -1608.405} C_VEL
LIN {X 0,Y 587.6,Z 807.613,A -85,B 0,C 180,E1 -1608.888,E2 -1608.888} C_VEL
LIN {X 0,Y 587.513,Z 819.013,A -85,B 0,C 180,E1 -1609.488,E2 -1609.488} C_VEL
LIN {X 0,Y 587.411,Z 829.484,A -85,B 0,C 180,E1 -1610.183,E2 -1610.183} C_VEL
LIN {X 0,Y 587.344,Z 840.029,A -85,B 0,C 180,E1 -1611.05,E2 -1611.05} C_VEL
LIN {X 0,Y 587.3,Z 848.594,A -85,B 0,C 180,E1 -1611.916,E2 -1611.916} C_VEL
LIN {X 0,Y 587.248,Z 856.909,A -85,B 0,C 180,E1 -1612.953,E2 -1612.953} C_VEL
LIN {X 0,Y 587.218,Z 863.61,A -85,B 0,C 180,E1 -1613.988,E2 -1613.988} C_VEL
LIN {X 0,Y 587.147,Z 869.755,A -85,B 0,C 180,E1 -1615.193,E2 -1615.193} C_VEL
LIN {X 0,Y 587.212,Z 873.745,A -85,B 0,C 180,E1 -1616.225,E2 -1616.225} C_VEL
LIN {X 0,Y 587.133,Z 876.694,A -85,B 0,C 180,E1 -1617.255,E2 -1617.255} C_VEL
LIN {X 0,Y 587.139,Z 878.127,A -85,B 0,C 180,E1 -1617.941,E2 -1617.941} C_VEL
LIN {X 0,Y 587.141,Z 879.753,A -85,B 0,C 180,E1 -1619.313,E2 -1619.313} C_VEL
LIN {X 0,Y 587.137,Z 879.996,A -85,B 0,C 180,E1 -1619.999,E2 -1619.999} C_VEL
LIN {X 0,Y 587.14,Z 879.815,A -85,B 0,C 180,E1 -1620.685,E2 -1620.685} C_VEL
LIN {X 0,Y 587.139,Z 878.275,A -85,B 0,C 180,E1 -1622.057,E2 -1622.057} C_VEL
LIN {X 0,Y 587.133,Z 876.915,A -85,B 0,C 180,E1 -1622.744,E2 -1622.744} C_VEL
LIN {X 0,Y 587.213,Z 874.038,A -85,B 0,C 180,E1 -1623.774,E2 -1623.774} C_VEL
LIN {X 0,Y 587.147,Z 870.139,A -85,B 0,C 180,E1 -1624.806,E2 -1624.806} C_VEL
LIN {X 0,Y 587.229,Z 865.108,A -85,B 0,C 180,E1 -1625.838,E2 -1625.838} C_VEL
LIN {X 0,Y 587.229,Z 858.789,A -85,B 0,C 180,E1 -1626.873,E2 -1626.873} C_VEL
LIN {X 0,Y 587.287,Z 850.871,A -85,B 0,C 180,E1 -1627.909,E2 -1627.909} C_VEL
LIN {X 0,Y 587.343,Z 841.026,A -85,B 0,C 180,E1 -1628.948,E2 -1628.948} C_VEL
LIN {X 0,Y 587.421,Z 830.705,A -85,B 0,C 180,E1 -1629.815,E2 -1629.815} C_VEL
LIN {X 0,Y 587.514,Z 819.082,A -85,B 0,C 180,E1 -1630.597,E2 -1630.597} C_VEL
LIN {X 0,Y 587.561,Z 808.441,A -85,B 0,C 180,E1 -1631.164,E2 -1631.164} C_VEL
LIN {X 0,Y 587.57,Z 796.757,A -85,B 0,C 180,E1 -1631.646,E2 -1631.646} C_VEL
LIN {X 0,Y 587.697,Z 783.438,A -85,B 0,C 180,E1 -1632.035,E2 -1632.035} C_VEL
LIN {X 0,Y 587.488,Z 778.761,A -85,B 0,C 180,E1 -1632.141,E2 -1632.141} C_VEL
LIN {X 0,Y 587.15,Z 776.673,A -85,B 0,C 180,E1 -1632.2,E2 -1632.2} C_VEL
LIN {X 0,Y 587.136,Z 773.672,A -85,B 0,C 180,E1 -1634.401,E2 -1634.401} C_VEL
LIN {X 0,Y 586.442,Z 772.926,A -85,B 0,C 180,E1 -1634.969,E2 -1634.969} C_VEL
LIN {X 0,Y 583.566,Z 771.788,A -85,B 0,C 180,E1 -1635.892,E2 -1635.892} C_VEL
LIN {X 0,Y 581.152,Z 770.889,A -85,B 0,C 180,E1 -1636.634,E2 -1636.634} C_VEL
LIN {X 0,Y 580.118,Z 770.171,A -85,B 0,C 180,E1 -1637.207,E2 -1637.207} C_VEL
LIN {X 0,Y 580.035,Z 769.918,A -85,B 0,C 180,E1 -1637.401,E2 -1637.401} C_VEL
LIN {X 0,Y 580.051,Z 766.729,A -85,B 0,C 180,E1 -1639.83,E2 -1639.83} C_VEL
LIN {X 0,Y 580.044,Z 763.845,A -85,B 0,C 180,E1 -1642.061,E2 -1642.061} C_VEL
LIN {X 0,Y 580.094,Z 760.512,A -85,B 0,C 180,E1 -1644.681,E2 -1644.681} C_VEL
LIN {X 0,Y 580.085,Z 757.115,A -85,B 0,C 180,E1 -1647.411,E2 -1647.411} C_VEL
LIN {X 0,Y 580.088,Z 754.23,A -85,B 0,C 180,E1 -1649.783,E2 -1649.783} C_VEL
LIN {X 0,Y 580.131,Z 751.378,A -85,B 0,C 180,E1 -1652.21,E2 -1652.21} C_VEL
LIN {X 0,Y 580.158,Z 749.525,A -85,B 0,C 180,E1 -1653.864,E2 -1653.864} C_VEL
LIN {X 0,Y 580.224,Z 749.209,A -85,B 0,C 180,E1 -1655.548,E2 -1655.548} C_VEL
LIN {X 0,Y 580.281,Z 749.197,A -85,B 0,C 180,E1 -1658.146,E2 -1658.146} C_VEL
LIN {X 0,Y 580.294,Z 749.199,A -85,B 0,C 180,E1 -1660.843,E2 -1660.843} C_VEL
LIN {X 0,Y 580.268,Z 749.203,A -85,B 0,C 180,E1 -1663.657,E2 -1663.657} C_VEL
LIN {X 0,Y 580.272,Z 749.198,A -85,B 0,C 180,E1 -1666.608,E2 -1666.608} C_VEL
LIN {X 0,Y 580.291,Z 749.202,A -85,B 0,C 180,E1 -1669.156,E2 -1669.156} C_VEL
LIN {X 0,Y 580.28,Z 749.2,A -85,B 0,C 180,E1 -1671.927,E2 -1671.927} C_VEL
LIN {X 0,Y 580.244,Z 749.201,A -85,B 0,C 180,E1 -1674.452,E2 -1674.452} C_VEL
LIN {X 0,Y 580.281,Z 749.199,A -85,B 0,C 180,E1 -1676.974,E2 -1676.974} C_VEL
LIN {X 0,Y 580.278,Z 749.205,A -85,B 0,C 180,E1 -1679.424,E2 -1679.424} C_VEL
LIN {X 0,Y 580.251,Z 749.203,A -85,B 0,C 180,E1 -1682.148,E2 -1682.148} C_VEL
LIN {X 0,Y 580.275,Z 749.198,A -85,B 0,C 180,E1 -1684.919,E2 -1684.919} C_VEL
LIN {X 0,Y 580.255,Z 749.206,A -85,B 0,C 180,E1 -1687.947,E2 -1687.947} C_VEL
LIN {X 0,Y 580.285,Z 749.196,A -85,B 0,C 180,E1 -1690.913,E2 -1690.913} C_VEL
LIN {X 0,Y 580.254,Z 749.21,A -85,B 0,C 180,E1 -1693.825,E2 -1693.825} C_VEL
LIN {X 0,Y 580.307,Z 749.201,A -85,B 0,C 180,E1 -1695.983,E2 -1695.983} C_VEL
LIN {X 0,Y 580.295,Z 749.195,A -85,B 0,C 180,E1 -1698.827,E2 -1698.827} C_VEL
LIN {X 0,Y 580.292,Z 749.201,A -85,B 0,C 180,E1 -1701.643,E2 -1701.643} C_VEL
LIN {X 0,Y 580.283,Z 749.199,A -85,B 0,C 180,E1 -1704.44,E2 -1704.44} C_VEL
LIN {X 0,Y 580.291,Z 749.195,A -85,B 0,C 180,E1 -1707.223,E2 -1707.223} C_VEL
LIN {X 0,Y 580.339,Z 749.199,A -85,B 0,C 180,E1 -1710,E2 -1710} C_VEL
LIN {X 0,Y 580.289,Z 749.196,A -85,B 0,C 180,E1 -1712.777,E2 -1712.777} C_VEL
LIN {X 0,Y 580.275,Z 749.199,A -85,B 0,C 180,E1 -1715.56,E2 -1715.56} C_VEL
LIN {X 0,Y 580.279,Z 749.204,A -85,B 0,C 180,E1 -1718.357,E2 -1718.357} C_VEL
LIN {X 0,Y 580.256,Z 749.199,A -85,B 0,C 180,E1 -1721.174,E2 -1721.174} C_VEL
LIN {X 0,Y 580.297,Z 749.201,A -85,B 0,C 180,E1 -1724.018,E2 -1724.018} C_VEL
LIN {X 0,Y 580.257,Z 749.201,A -85,B 0,C 180,E1 -1726.899,E2 -1726.899} C_VEL
LIN {X 0,Y 580.27,Z 749.2,A -85,B 0,C 180,E1 -1729.824,E2 -1729.824} C_VEL
LIN {X 0,Y 580.252,Z 749.205,A -85,B 0,C 180,E1 -1732.054,E2 -1732.054} C_VEL
LIN {X 0,Y 580.27,Z 749.199,A -85,B 0,C 180,E1 -1735.082,E2 -1735.082} C_VEL
LIN {X 0,Y 580.271,Z 749.203,A -85,B 0,C 180,E1 -1738.187,E2 -1738.187} C_VEL
LIN {X 0,Y 580.266,Z 749.206,A -85,B 0,C 180,E1 -1740.693,E2 -1740.693} C_VEL
LIN {X 0,Y 580.273,Z 749.198,A -85,B 0,C 180,E1 -1743.314,E2 -1743.314} C_VEL
LIN {X 0,Y 580.237,Z 749.202,A -85,B 0,C 180,E1 -1745.757,E2 -1745.757} C_VEL
LIN {X 0,Y 580.278,Z 749.2,A -85,B 0,C 180,E1 -1748.147,E2 -1748.147} C_VEL
LIN {X 0,Y 580.289,Z 749.203,A -85,B 0,C 180,E1 -1750.844,E2 -1750.844} C_VEL
LIN {X 0,Y 580.267,Z 749.198,A -85,B 0,C 180,E1 -1753.659,E2 -1753.659} C_VEL
LIN {X 0,Y 580.27,Z 749.206,A -85,B 0,C 180,E1 -1756.61,E2 -1756.61} C_VEL
LIN {X 0,Y 580.292,Z 749.2,A -85,B 0,C 180,E1 -1759.157,E2 -1759.157} C_VEL
LIN {X 0,Y 580.282,Z 749.197,A -85,B 0,C 180,E1 -1761.928,E2 -1761.928} C_VEL
LIN {X 0,Y 580.245,Z 749.205,A -85,B 0,C 180,E1 -1764.453,E2 -1764.453} C_VEL
LIN {X 0,Y 580.113,Z 749.228,A -85,B 0,C 180,E1 -1766.133,E2 -1766.133} C_VEL
LIN {X 0,Y 580.124,Z 752.179,A -85,B 0,C 180,E1 -1768.606,E2 -1768.606} C_VEL
LIN {X 0,Y 580.094,Z 755.083,A -85,B 0,C 180,E1 -1771.014,E2 -1771.014} C_VEL
LIN {X 0,Y 580.124,Z 758.374,A -85,B 0,C 180,E1 -1773.7,E2 -1773.7} C_VEL
LIN {X 0,Y 580.066,Z 761.808,A -85,B 0,C 180,E1 -1776.434,E2 -1776.434} C_VEL
LIN {X 0,Y 580.084,Z 765.651,A -85,B 0,C 180,E1 -1779.431,E2 -1779.431} C_VEL
LIN {X 0,Y 580.043,Z 769.494,A -85,B 0,C 180,E1 -1782.368,E2 -1782.368} C_VEL
LIN {X 0,Y 580.051,Z 772.377,A -85,B 0,C 180,E1 -1784.541,E2 -1784.541} C_VEL
LIN {X 0,Y 580.052,Z 775.259,A -85,B 0,C 180,E1 -1786.692,E2 -1786.692} C_VEL
LIN {X 0,Y 580.074,Z 776.671,A -85,B 0,C 180,E1 -1787.738,E2 -1787.738} C_VEL
LIN {X 0,Y 580.775,Z 782.355,A -85,B 0,C 180,E1 -1787.886,E2 -1787.886} C_VEL
LIN {X 0,Y 580.672,Z 794.129,A -85,B 0,C 180,E1 -1788.216,E2 -1788.216} C_VEL
LIN {X 0,Y 580.594,Z 805.682,A -85,B 0,C 180,E1 -1788.666,E2 -1788.666} C_VEL
LIN {X 0,Y 580.546,Z 817.55,A -85,B 0,C 180,E1 -1789.274,E2 -1789.274} C_VEL
LIN {X 0,Y 580.451,Z 828.343,A -85,B 0,C 180,E1 -1789.977,E2 -1789.977} C_VEL
LIN {X 0,Y 580.333,Z 838.104,A -85,B 0,C 180,E1 -1790.767,E2 -1790.767} C_VEL
LIN {X 0,Y 580.264,Z 846.996,A -85,B 0,C 180,E1 -1791.644,E2 -1791.644} C_VEL
LIN {X 0,Y 580.199,Z 854.335,A -85,B 0,C 180,E1 -1792.519,E2 -1792.519} C_VEL
LIN {X 0,Y 580.17,Z 860.345,A -85,B 0,C 180,E1 -1793.378,E2 -1793.378} C_VEL
LIN {X 0,Y 580.139,Z 866.43,A -85,B 0,C 180,E1 -1794.439,E2 -1794.439} C_VEL
LIN {X 0,Y 580.107,Z 871.177,A -85,B 0,C 180,E1 -1795.484,E2 -1795.484} C_VEL
LIN {X 0,Y 580.123,Z 874.815,A -85,B 0,C 180,E1 -1796.528,E2 -1796.528} C_VEL
LIN {X 0,Y 580.043,Z 876.689,A -85,B 0,C 180,E1 -1797.223,E2 -1797.223} C_VEL
LIN {X 0,Y 580.038,Z 878.133,A -85,B 0,C 180,E1 -1797.918,E2 -1797.918} C_VEL
LIN {X 0,Y 580.041,Z 879.754,A -85,B 0,C 180,E1 -1799.306,E2 -1799.306} C_VEL
LIN {X 0,Y 580.038,Z 879.997,A -85,B 0,C 180,E1 -1800.001,E2 -1800.001} C_VEL
LIN {X 0,Y 580.04,Z 879.811,A -85,B 0,C 180,E1 -1800.695,E2 -1800.695} C_VEL
LIN {X 0,Y 580.037,Z 878.276,A -85,B 0,C 180,E1 -1802.084,E2 -1802.084} C_VEL
LIN {X 0,Y 580.044,Z 876.889,A -85,B 0,C 180,E1 -1802.779,E2 -1802.779} C_VEL
LIN {X 0,Y 580.11,Z 874.013,A -85,B 0,C 180,E1 -1803.821,E2 -1803.821} C_VEL
LIN {X 0,Y 580.053,Z 870.112,A -85,B 0,C 180,E1 -1804.866,E2 -1804.866} C_VEL
LIN {X 0,Y 580.161,Z 865.085,A -85,B 0,C 180,E1 -1805.911,E2 -1805.911} C_VEL
LIN {X 0,Y 580.185,Z 857.553,A -85,B 0,C 180,E1 -1807.133,E2 -1807.133} C_VEL
LIN {X 0,Y 580.245,Z 849.366,A -85,B 0,C 180,E1 -1808.183,E2 -1808.183} C_VEL
LIN {X 0,Y 580.307,Z 840.968,A -85,B 0,C 180,E1 -1809.059,E2 -1809.059} C_VEL
LIN {X 0,Y 580.408,Z 830.68,A -85,B 0,C 180,E1 -1809.937,E2 -1809.937} C_VEL
LIN {X 0,Y 580.526,Z 819.063,A -85,B 0,C 180,E1 -1810.728,E2 -1810.728} C_VEL
LIN {X 0,Y 580.615,Z 807.424,A -85,B 0,C 180,E1 -1811.345,E2 -1811.345} C_VEL
LIN {X 0,Y 580.683,Z 795.411,A -85,B 0,C 180,E1 -1811.83,E2 -1811.83} C_VEL
LIN {X 0,Y 580.753,Z 783.301,A -85,B 0,C 180,E1 -1812.183,E2 -1812.183} C_VEL
LIN {X 0,Y 580.35,Z 778.552,A -85,B 0,C 180,E1 -1812.297,E2 -1812.297} C_VEL
LIN {X 0,Y 580.082,Z 776.67,A -85,B 0,C 180,E1 -1812.353,E2 -1812.353} C_VEL
LIN {X 0,Y 580.047,Z 773.456,A -85,B 0,C 180,E1 -1814.741,E2 -1814.741} C_VEL
LIN {X 0,Y 580.067,Z 770.572,A -85,B 0,C 180,E1 -1816.905,E2 -1816.905} C_VEL
LIN {X 0,Y 580.063,Z 766.727,A -85,B 0,C 180,E1 -1819.832,E2 -1819.832} C_VEL
LIN {X 0,Y 580.047,Z 763.843,A -85,B 0,C 180,E1 -1822.062,E2 -1822.062} C_VEL
LIN {X 0,Y 580.093,Z 760.512,A -85,B 0,C 180,E1 -1824.68,E2 -1824.68} C_VEL
LIN {X 0,Y 580.089,Z 757.113,A -85,B 0,C 180,E1 -1827.412,E2 -1827.412} C_VEL
LIN {X 0,Y 580.088,Z 754.228,A -85,B 0,C 180,E1 -1829.785,E2 -1829.785} C_VEL
LIN {X 0,Y 580.091,Z 751.139,A -85,B 0,C 180,E1 -1832.214,E2 -1832.214} C_VEL
LIN {X 0,Y 580.099,Z 749.607,A -85,B 0,C 180,E1 -1833.285,E2 -1833.285} C_VEL
LIN {X 0,Y 580.198,Z 749.217,A -85,B 0,C 180,E1 -1834.544,E2 -1834.544} C_VEL
LIN {X 0,Y 580.292,Z 749.205,A -85,B 0,C 180,E1 -1837.269,E2 -1837.269} C_VEL
LIN {X 0,Y 580.297,Z 749.196,A -85,B 0,C 180,E1 -1840.271,E2 -1840.271} C_VEL
LIN {X 0,Y 580.273,Z 749.203,A -85,B 0,C 180,E1 -1843.39,E2 -1843.39} C_VEL
LIN {X 0,Y 580.283,Z 749.198,A -85,B 0,C 180,E1 -1846.342,E2 -1846.342} C_VEL
LIN {X 0,Y 580.302,Z 749.203,A -85,B 0,C 180,E1 -1849.157,E2 -1849.157} C_VEL
LIN {X 0,Y 580.295,Z 749.199,A -85,B 0,C 180,E1 -1851.927,E2 -1851.927} C_VEL
LIN {X 0,Y 580.327,Z 749.351,A -85,B 0,C 180,E1 -1853.505,E2 -1853.505} C_VEL
LIN {X 0,Y 580.766,Z 753.571,A -85,B 0,C 180,E1 -1854.913,E2 -1854.913} C_VEL
LIN {X 0,Y 580.709,Z 762.841,A -85,B 0,C 180,E1 -1857.825,E2 -1857.825} C_VEL
LIN {X 0,Y 580.568,Z 772.136,A -85,B 0,C 180,E1 -1860.644,E2 -1860.644} C_VEL
LIN {X 0,Y 580.496,Z 781.394,A -85,B 0,C 180,E1 -1863.387,E2 -1863.387} C_VEL
LIN {X 0,Y 580.421,Z 790.661,A -85,B 0,C 180,E1 -1866.069,E2 -1866.069} C_VEL
LIN {X 0,Y 580.323,Z 800.405,A -85,B 0,C 180,E1 -1868.83,E2 -1868.83} C_VEL
LIN {X 0,Y 580.253,Z 810.52,A -85,B 0,C 180,E1 -1871.644,E2 -1871.644} C_VEL
LIN {X 0,Y 580.193,Z 821.111,A -85,B 0,C 180,E1 -1874.544,E2 -1874.544} C_VEL
LIN {X 0,Y 580.169,Z 831.703,A -85,B 0,C 180,E1 -1877.406,E2 -1877.406} C_VEL
LIN {X 0,Y 580.149,Z 832.53,A -85,B 0,C 180,E1 -1877.627,E2 -1877.627} C_VEL
LIN {X 0,Y 580.795,Z 838.227,A -85,B 0,C 180,E1 -1877.752,E2 -1877.752} C_VEL
LIN {X 0,Y 580.743,Z 851.495,A -85,B 0,C 180,E1 -1878.083,E2 -1878.083} C_VEL
LIN {X 0,Y 580.611,Z 863.576,A -85,B 0,C 180,E1 -1878.526,E2 -1878.526} C_VEL
LIN {X 0,Y 580.552,Z 875.209,A -85,B 0,C 180,E1 -1879.097,E2 -1879.097} C_VEL
LIN {X 0,Y 580.448,Z 886.477,A -85,B 0,C 180,E1 -1879.8,E2 -1879.8} C_VEL
LIN {X 0,Y 580.352,Z 896.646,A -85,B 0,C 180,E1 -1880.591,E2 -1880.591} C_VEL
LIN {X 0,Y 580.279,Z 905.787,A -85,B 0,C 180,E1 -1881.468,E2 -1881.468} C_VEL
LIN {X 0,Y 580.199,Z 914.69,A -85,B 0,C 180,E1 -1882.518,E2 -1882.518} C_VEL
LIN {X 0,Y 580.12,Z 921.468,A -85,B 0,C 180,E1 -1883.505,E2 -1883.505} C_VEL
LIN {X 0,Y 580.139,Z 926.68,A -85,B 0,C 180,E1 -1884.438,E2 -1884.438} C_VEL
LIN {X 0,Y 580.108,Z 931.371,A -85,B 0,C 180,E1 -1885.483,E2 -1885.483} C_VEL
LIN {X 0,Y 580.123,Z 934.956,A -85,B 0,C 180,E1 -1886.527,E2 -1886.527} C_VEL
LIN {X 0,Y 580.043,Z 936.809,A -85,B 0,C 180,E1 -1887.222,E2 -1887.222} C_VEL
LIN {X 0,Y 580.038,Z 938.201,A -85,B 0,C 180,E1 -1887.917,E2 -1887.917} C_VEL
LIN {X 0,Y 580.04,Z 939.784,A -85,B 0,C 180,E1 -1889.306,E2 -1889.306} C_VEL
LIN {X 0,Y 580.037,Z 940,A -85,B 0,C 180,E1 -1890,E2 -1890} C_VEL
LIN {X 0,Y 580.047,Z 939.185,A -85,B 0,C 180,E1 -1891.389,E2 -1891.389} C_VEL
LIN {X 0,Y 580.038,Z 938.201,A -85,B 0,C 180,E1 -1892.083,E2 -1892.083} C_VEL
LIN {X 0,Y 580.043,Z 936.81,A -85,B 0,C 180,E1 -1892.778,E2 -1892.778} C_VEL
LIN {X 0,Y 580.109,Z 933.896,A -85,B 0,C 180,E1 -1893.821,E2 -1893.821} C_VEL
LIN {X 0,Y 580.054,Z 929.949,A -85,B 0,C 180,E1 -1894.865,E2 -1894.865} C_VEL
LIN {X 0,Y 580.139,Z 923.877,A -85,B 0,C 180,E1 -1896.085,E2 -1896.085} C_VEL
LIN {X 0,Y 580.184,Z 917.236,A -85,B 0,C 180,E1 -1897.132,E2 -1897.132} C_VEL
LIN {X 0,Y 580.25,Z 908.989,A -85,B 0,C 180,E1 -1898.182,E2 -1898.182} C_VEL
LIN {X 0,Y 580.308,Z 900.537,A -85,B 0,C 180,E1 -1899.058,E2 -1899.058} C_VEL
LIN {X 0,Y 580.414,Z 890.094,A -85,B 0,C 180,E1 -1899.936,E2 -1899.936} C_VEL
LIN {X 0,Y 580.519,Z 879.758,A -85,B 0,C 180,E1 -1900.639,E2 -1900.639} C_VEL
LIN {X 0,Y 580.573,Z 868.493,A -85,B 0,C 180,E1 -1901.252,E2 -1901.252} C_VEL
LIN {X 0,Y 580.674,Z 856.765,A -85,B 0,C 180,E1 -1901.741,E2 -1901.741} C_VEL
LIN {X 0,Y 580.777,Z 843.348,A -85,B 0,C 180,E1 -1902.137,E2 -1902.137} C_VEL
LIN {X 0,Y 580.55,Z 835.159,A -85,B 0,C 180,E1 -1902.311,E2 -1902.311} C_VEL
LIN {X 0,Y 580.149,Z 832.53,A -85,B 0,C 180,E1 -1902.373,E2 -1902.373} C_VEL
LIN {X 0,Y 580.216,Z 822.435,A -85,B 0,C 180,E1 -1905.095,E2 -1905.095} C_VEL
LIN {X 0,Y 580.254,Z 811.844,A -85,B 0,C 180,E1 -1907.99,E2 -1907.99} C_VEL
LIN {X 0,Y 580.345,Z 801.491,A -85,B 0,C 180,E1 -1910.864,E2 -1910.864} C_VEL
LIN {X 0,Y 580.408,Z 791.985,A -85,B 0,C 180,E1 -1913.553,E2 -1913.553} C_VEL
LIN {X 0,Y 580.486,Z 782.219,A -85,B 0,C 180,E1 -1916.372,E2 -1916.372} C_VEL
LIN {X 0,Y 580.526,Z 773.451,A -85,B 0,C 180,E1 -1918.964,E2 -1918.964} C_VEL
LIN {X 0,Y 580.671,Z 764.316,A -85,B 0,C 180,E1 -1921.728,E2 -1921.728} C_VEL
LIN {X 0,Y 580.716,Z 756.177,A -85,B 0,C 180,E1 -1924.223,E2 -1924.223} C_VEL
LIN {X 0,Y 580.673,Z 751.419,A -85,B 0,C 180,E1 -1925.814,E2 -1925.814} C_VEL
LIN {X 0,Y 580.325,Z 749.201,A -85,B 0,C 180,E1 -1926.686,E2 -1926.686} C_VEL
LIN {X 0,Y 580.302,Z 749.204,A -85,B 0,C 180,E1 -1929.185,E2 -1929.185} C_VEL
LIN {X 0,Y 580.294,Z 749.198,A -85,B 0,C 180,E1 -1931.768,E2 -1931.768} C_VEL
LIN {X 0,Y 580.266,Z 749.204,A -85,B 0,C 180,E1 -1934.626,E2 -1934.626} C_VEL
LIN {X 0,Y 580.267,Z 749.206,A -85,B 0,C 180,E1 -1937.292,E2 -1937.292} C_VEL
LIN {X 0,Y 580.288,Z 749.198,A -85,B 0,C 180,E1 -1940.066,E2 -1940.066} C_VEL
LIN {X 0,Y 580.282,Z 749.206,A -85,B 0,C 180,E1 -1943.068,E2 -1943.068} C_VEL
LIN {X 0,Y 580.213,Z 749.216,A -85,B 0,C 180,E1 -1945.454,E2 -1945.454} C_VEL
LIN {X 0,Y 580.133,Z 751.695,A -85,B 0,C 180,E1 -1947.997,E2 -1947.997} C_VEL
LIN {X 0,Y 580.088,Z 754.12,A -85,B 0,C 180,E1 -1950.215,E2 -1950.215} C_VEL
LIN {X 0,Y 580.089,Z 757.002,A -85,B 0,C 180,E1 -1952.588,E2 -1952.588} C_VEL
LIN {X 0,Y 580.117,Z 760.845,A -85,B 0,C 180,E1 -1955.675,E2 -1955.675} C_VEL
LIN {X 0,Y 580.064,Z 764.688,A -85,B 0,C 180,E1 -1958.686,E2 -1958.686} C_VEL
LIN {X 0,Y 580.071,Z 767.583,A -85,B 0,C 180,E1 -1960.915,E2 -1960.915} C_VEL
LIN {X 0,Y 580.082,Z 771.414,A -85,B 0,C 180,E1 -1963.819,E2 -1963.819} C_VEL
LIN {X 0,Y 580.054,Z 775.257,A -85,B 0,C 180,E1 -1966.69,E2 -1966.69} C_VEL
LIN {X 0,Y 580.06,Z 776.669,A -85,B 0,C 180,E1 -1967.736,E2 -1967.736} C_VEL
LIN {X 0,Y 580.761,Z 782.382,A -85,B 0,C 180,E1 -1967.884,E2 -1967.884} C_VEL
LIN {X 0,Y 580.683,Z 795.433,A -85,B 0,C 180,E1 -1968.259,E2 -1968.259} C_VEL
LIN {X 0,Y 580.625,Z 807.299,A -85,B 0,C 180,E1 -1968.738,E2 -1968.738} C_VEL
LIN {X 0,Y 580.535,Z 819.021,A -85,B 0,C 180,E1 -1969.361,E2 -1969.361} C_VEL
LIN {X 0,Y 580.385,Z 830.654,A -85,B 0,C 180,E1 -1970.151,E2 -1970.151} C_VEL
LIN {X 0,Y 580.308,Z 840.035,A -85,B 0,C 180,E1 -1970.941,E2 -1970.941} C_VEL
LIN {X 0,Y 580.251,Z 848.599,A -85,B 0,C 180,E1 -1971.817,E2 -1971.817} C_VEL
LIN {X 0,Y 580.186,Z 856.914,A -85,B 0,C 180,E1 -1972.867,E2 -1972.867} C_VEL
LIN {X 0,Y 580.14,Z 863.613,A -85,B 0,C 180,E1 -1973.915,E2 -1973.915} C_VEL
LIN {X 0,Y 580.054,Z 869.758,A -85,B 0,C 180,E1 -1975.134,E2 -1975.134} C_VEL
LIN {X 0,Y 580.109,Z 873.747,A -85,B 0,C 180,E1 -1976.179,E2 -1976.179} C_VEL
LIN {X 0,Y 580.044,Z 876.696,A -85,B 0,C 180,E1 -1977.221,E2 -1977.221} C_VEL
LIN {X 0,Y 580.039,Z 878.127,A -85,B 0,C 180,E1 -1977.916,E2 -1977.916} C_VEL
LIN {X 0,Y 580.041,Z 879.754,A -85,B 0,C 180,E1 -1979.305,E2 -1979.305} C_VEL
LIN {X 0,Y 580.038,Z 879.996,A -85,B 0,C 180,E1 -1979.999,E2 -1979.999} C_VEL
LIN {X 0,Y 580.04,Z 879.815,A -85,B 0,C 180,E1 -1980.694,E2 -1980.694} C_VEL
LIN {X 0,Y 580.038,Z 878.274,A -85,B 0,C 180,E1 -1982.082,E2 -1982.082} C_VEL
LIN {X 0,Y 580.044,Z 876.913,A -85,B 0,C 180,E1 -1982.777,E2 -1982.777} C_VEL
LIN {X 0,Y 580.11,Z 874.036,A -85,B 0,C 180,E1 -1983.82,E2 -1983.82} C_VEL
LIN {X 0,Y 580.053,Z 870.137,A -85,B 0,C 180,E1 -1984.865,E2 -1984.865} C_VEL
LIN {X 0,Y 580.162,Z 865.105,A -85,B 0,C 180,E1 -1985.909,E2 -1985.909} C_VEL
LIN {X 0,Y 580.157,Z 858.785,A -85,B 0,C 180,E1 -1986.957,E2 -1986.957} C_VEL
LIN {X 0,Y 580.242,Z 850.867,A -85,B 0,C 180,E1 -1988.006,E2 -1988.006} C_VEL
LIN {X 0,Y 580.308,Z 841.02,A -85,B 0,C 180,E1 -1989.058,E2 -1989.058} C_VEL
LIN {X 0,Y 580.421,Z 830.699,A -85,B 0,C 180,E1 -1989.935,E2 -1989.935} C_VEL
LIN {X 0,Y 580.523,Z 819.072,A -85,B 0,C 180,E1 -1990.726,E2 -1990.726} C_VEL
LIN {X 0,Y 580.602,Z 807.611,A -85,B 0,C 180,E1 -1991.338,E2 -1991.338} C_VEL
LIN {X 0,Y 580.651,Z 795.646,A -85,B 0,C 180,E1 -1991.825,E2 -1991.825} C_VEL
LIN {X 0,Y 580.775,Z 782.5,A -85,B 0,C 180,E1 -1992.203,E2 -1992.203} C_VEL
LIN {X 0,Y 580.083,Z 776.672,A -85,B 0,C 180,E1 -1992.351,E2 -1992.351} C_VEL
LIN {X 0,Y 580.041,Z 773.458,A -85,B 0,C 180,E1 -1994.74,E2 -1994.74} C_VEL
LIN {X 0,Y 580.035,Z 769.918,A -85,B 0,C 180,E1 -1997.401,E2 -1997.401} C_VEL
LIN {X 0,Y 579.367,Z 769.187,A -85,B 0,C 180,E1 -1997.976,E2 -1997.976} C_VEL
LIN {X 0,Y 576.501,Z 768.087,A -85,B 0,C 180,E1 -1998.911,E2 -1998.911} C_VEL
LIN {X 0,Y 574.082,Z 767.221,A -85,B 0,C 180,E1 -1999.663,E2 -1999.663} C_VEL
LIN {X 0,Y 573.048,Z 766.522,A -85,B 0,C 180,E1 -2000.244,E2 -2000.244} C_VEL
LIN {X 0,Y 572.967,Z 766.274,A -85,B 0,C 180,E1 -2000.44,E2 -2000.44} C_VEL
LIN {X 0,Y 572.987,Z 762.883,A -85,B 0,C 180,E1 -2003.109,E2 -2003.109} C_VEL
LIN {X 0,Y 573.001,Z 759.998,A -85,B 0,C 180,E1 -2005.421,E2 -2005.421} C_VEL
LIN {X 0,Y 573.017,Z 756.865,A -85,B 0,C 180,E1 -2007.984,E2 -2007.984} C_VEL
LIN {X 0,Y 573.041,Z 753.298,A -85,B 0,C 180,E1 -2011.003,E2 -2011.003} C_VEL
LIN {X 0,Y 573.069,Z 750.528,A -85,B 0,C 180,E1 -2013.494,E2 -2013.494} C_VEL
LIN {X 0,Y 573.152,Z 750.095,A -85,B 0,C 180,E1 -2014.759,E2 -2014.759} C_VEL
LIN {X 0,Y 573.248,Z 750.083,A -85,B 0,C 180,E1 -2017.165,E2 -2017.165} C_VEL
LIN {X 0,Y 573.234,Z 750.08,A -85,B 0,C 180,E1 -2019.607,E2 -2019.607} C_VEL
LIN {X 0,Y 573.236,Z 750.076,A -85,B 0,C 180,E1 -2022.641,E2 -2022.641} C_VEL
LIN {X 0,Y 573.23,Z 750.081,A -85,B 0,C 180,E1 -2025.666,E2 -2025.666} C_VEL
LIN {X 0,Y 573.222,Z 750.076,A -85,B 0,C 180,E1 -2028.542,E2 -2028.542} C_VEL
LIN {X 0,Y 573.235,Z 750.083,A -85,B 0,C 180,E1 -2031.298,E2 -2031.298} C_VEL
LIN {X 0,Y 573.206,Z 750.081,A -85,B 0,C 180,E1 -2034.018,E2 -2034.018} C_VEL
LIN {X 0,Y 573.223,Z 750.076,A -85,B 0,C 180,E1 -2036.515,E2 -2036.515} C_VEL
LIN {X 0,Y 573.215,Z 750.08,A -85,B 0,C 180,E1 -2039.118,E2 -2039.118} C_VEL
LIN {X 0,Y 573.222,Z 750.084,A -85,B 0,C 180,E1 -2041.435,E2 -2041.435} C_VEL
LIN {X 0,Y 573.225,Z 750.076,A -85,B 0,C 180,E1 -2044.588,E2 -2044.588} C_VEL
LIN {X 0,Y 573.22,Z 750.087,A -85,B 0,C 180,E1 -2047.661,E2 -2047.661} C_VEL
LIN {X 0,Y 573.256,Z 750.072,A -85,B 0,C 180,E1 -2050.67,E2 -2050.67} C_VEL
LIN {X 0,Y 573.23,Z 750.083,A -85,B 0,C 180,E1 -2053.621,E2 -2053.621} C_VEL
LIN {X 0,Y 573.258,Z 750.082,A -85,B 0,C 180,E1 -2055.807,E2 -2055.807} C_VEL
LIN {X 0,Y 573.253,Z 750.072,A -85,B 0,C 180,E1 -2058.745,E2 -2058.745} C_VEL
LIN {X 0,Y 573.235,Z 750.078,A -85,B 0,C 180,E1 -2061.54,E2 -2061.54} C_VEL
